  [197] = {x=-25.429863, y=27.236716, z=96.648372, rx=-178.000688, ry=-0.000306, rz=-0.000289, shoulder=lefty, elbow=epositive, wrist=wpositive, fatherId=frmaster[2]}
  [198] = {x=-24.431312, y=27.249472, z=96.640619, rx=-177.999992, ry=-0.000305, rz=0.000037, shoulder=lefty, elbow=epositive, wrist=wpositive, fatherId=frmaster[2]}
  [199] = {x=-23.439357, y=27.256646, z=96.642496, rx=-178.000278, ry=-0.00008, rz=0.00033, shoulder=lefty, elbow=epositive, wrist=wpositive, fatherId=frmaster[2]}
  [200] = {x=-22.438851, y=27.268013, z=96.64425, rx=-178.000546, ry=0.000117, rz=-0.000381, shoulder=lefty, elbow=epositive, wrist=wpositive, fatherId=frmaster[2]}
  [201] = {x=-21.43819, y=27.28289, z=96.645991, rx=-177.999822, ry=0.000137, rz=-0.000095, shoulder=lefty, elbow=epositive, wrist=wpositive, fatherId=frmaster[2]}
  [202] = {x=-20.443726, y=27.289844, z=96.648903, rx=-178.001063, ry=0.000565, rz=0.000171, shoulder=lefty, elbow=epositive, wrist=wpositive, fatherId=frmaster[2]}
  [203] = {x=-19.450271, y=27.300156, z=96.643398, rx=-178.000499, ry=-0.00027, rz=0.00003, shoulder=lefty, elbow=epositive, wrist=wpositive, fatherId=frmaster[2]}
  [204] = {x=-18.446659, y=27.31259, z=96.642606, rx=-177.999749, ry=-0.000237, rz=-0.000711, shoulder=lefty, elbow=epositive, wrist=wpositive, fatherId=frmaster[2]}
  [205] = {x=-17.450599, y=27.324153, z=96.641778, rx=-177.999982, ry=0.000019, rz=-0.000456, shoulder=lefty, elbow=epositive, wrist=wpositive, fatherId=frmaster[2]}
  [206] = {x=-16.452954, y=27.332175, z=96.642123, rx=-178.000204, ry=0.000286, rz=-0.000221, shoulder=lefty, elbow=epositive, wrist=wpositive, fatherId=frmaster[2]}
  [207] = {x=-15.456767, y=27.345858, z=96.637596, rx=-177.999612, ry=-0.000534, rz=-0.00039, shoulder=lefty, elbow=epositive, wrist=wpositive, fatherId=frmaster[2]}
  [208] = {x=-14.4578, y=27.356168, z=96.642655, rx=-177.999817, ry=-0.000253, rz=-0.000178, shoulder=lefty, elbow=epositive, wrist=wpositive, fatherId=frmaster[2]}
  [209] = {x=-13.46591, y=27.363257, z=96.644106, rx=-178.00002, ry=0.000066, rz=0.000029, shoulder=lefty, elbow=epositive, wrist=wpositive, fatherId=frmaster[2]}
  [210] = {x=-12.465449, y=27.37475, z=96.645422, rx=-178.000206, ry=0.000355, rz=0.000232, shoulder=lefty, elbow=epositive, wrist=wpositive, fatherId=frmaster[2]}
  [211] = {x=-11.465766, y=27.388433, z=96.638237, rx=-177.999587, ry=-0.000451, rz=-0.000966, shoulder=lefty, elbow=epositive, wrist=wpositive, fatherId=frmaster[2]}
  [212] = {x=-10.471416, y=27.396685, z=96.64071, rx=-177.999763, ry=-0.000114, rz=0.000213, shoulder=lefty, elbow=epositive, wrist=wpositive, fatherId=frmaster[2]}
  [213] = {x=-9.476659, y=27.407266, z=96.643115, rx=-177.99993, ry=0.000228, rz=0.000387, shoulder=lefty, elbow=epositive, wrist=wpositive, fatherId=frmaster[2]}
  [214] = {x=-8.473698, y=27.418659, z=96.641745, rx=-178.000267, ry=-0.000352, rz=-0.000853, shoulder=lefty, elbow=epositive, wrist=wpositive, fatherId=frmaster[2]}
  [215] = {x=-7.476841, y=27.428148, z=96.645231, rx=-178.000415, ry=0.000004, rz=-0.000703, shoulder=lefty, elbow=epositive, wrist=wpositive, fatherId=frmaster[2]}
  [216] = {x=-6.479573, y=27.439988, z=96.648645, rx=-178.000553, ry=0.000365, rz=-0.000557, shoulder=lefty, elbow=epositive, wrist=wpositive, fatherId=frmaster[2]}
  [217] = {x=-5.482244, y=27.450503, z=96.648342, rx=-178.000876, ry=-0.000161, rz=-0.000826, shoulder=lefty, elbow=epositive, wrist=wpositive, fatherId=frmaster[2]}
  [218] = {x=-4.49109, y=27.459137, z=96.644439, rx=-178.000029, ry=0.000027, rz=0.000311, shoulder=lefty, elbow=epositive, wrist=wpositive, fatherId=frmaster[2]}
  [219] = {x=-3.491358, y=27.47236, z=96.640386, rx=-177.999165, ry=0.000182, rz=0.000444, shoulder=lefty, elbow=epositive, wrist=wpositive, fatherId=frmaster[2]}
  [220] = {x=-2.491458, y=27.484219, z=96.641061, rx=-177.999465, ry=-0.000328, rz=-0.000853, shoulder=lefty, elbow=epositive, wrist=wpositive, fatherId=frmaster[2]}
  [221] = {x=-1.497362, y=27.492926, z=96.646554, rx=-178.000541, ry=0.000317, rz=0.000238, shoulder=lefty, elbow=epositive, wrist=wpositive, fatherId=frmaster[2]}
  [222] = {x=-0.495266, y=27.503824, z=96.648283, rx=-178.000826, ry=-0.000176, rz=-0.001082, shoulder=lefty, elbow=epositive, wrist=wpositive, fatherId=frmaster[2]}
  [223] = {x=0.500089, y=27.515119, z=96.641527, rx=-177.999935, ry=0.000028, rz=0.000016, shoulder=lefty, elbow=epositive, wrist=wpositive, fatherId=frmaster[2]}
  [224] = {x=1.495371, y=27.526248, z=96.639538, rx=-177.99924, ry=-0.000651, rz=-0.000313, shoulder=lefty, elbow=epositive, wrist=wpositive, fatherId=frmaster[2]}
  [225] = {x=2.49304, y=27.536538, z=96.642297, rx=-177.999304, ry=-0.000205, rz=-0.000256, shoulder=lefty, elbow=epositive, wrist=wpositive, fatherId=frmaster[2]}
  [226] = {x=3.491932, y=27.545823, z=96.641306, rx=-177.999358, ry=0.000245, rz=-0.000205, shoulder=lefty, elbow=epositive, wrist=wpositive, fatherId=frmaster[2]}
  [227] = {x=4.490166, y=27.557254, z=96.640215, rx=-177.999614, ry=-0.00019, rz=-0.000562, shoulder=lefty, elbow=epositive, wrist=wpositive, fatherId=frmaster[2]}
  [228] = {x=5.482361, y=27.566672, z=96.643983, rx=-177.999657, ry=0.000308, rz=0.000462, shoulder=lefty, elbow=epositive, wrist=wpositive, fatherId=frmaster[2]}
  [229] = {x=6.482875, y=27.57725, z=96.643913, rx=-177.999897, ry=-0.000112, rz=0.00008, shoulder=lefty, elbow=epositive, wrist=wpositive, fatherId=frmaster[2]}
  [230] = {x=7.476743, y=27.588075, z=96.643826, rx=-177.999922, ry=0.000394, rz=0.000095, shoulder=lefty, elbow=epositive, wrist=wpositive, fatherId=frmaster[2]}
  [231] = {x=8.478648, y=27.6013, z=96.639929, rx=-177.999177, ry=-0.000259, rz=-0.000296, shoulder=lefty, elbow=epositive, wrist=wpositive, fatherId=frmaster[2]}
  [232] = {x=9.473739, y=27.611047, z=96.640839, rx=-177.999403, ry=-0.000629, rz=-0.000709, shoulder=lefty, elbow=epositive, wrist=wpositive, fatherId=frmaster[2]}
  [233] = {x=10.471276, y=27.620049, z=96.646501, rx=-178.000369, ry=0.000144, rz=0.000258, shoulder=lefty, elbow=epositive, wrist=wpositive, fatherId=frmaster[2]}
  [234] = {x=11.467775, y=27.632457, z=96.64357, rx=-177.999611, ry=-0.000461, rz=-0.000163, shoulder=lefty, elbow=epositive, wrist=wpositive, fatherId=frmaster[2]}
  [235] = {x=12.467578, y=27.640793, z=96.641696, rx=-177.999588, ry=0.000076, rz=-0.000206, shoulder=lefty, elbow=epositive, wrist=wpositive, fatherId=frmaster[2]}
  [236] = {x=13.465879, y=27.654652, z=96.643403, rx=-177.999783, ry=-0.000272, rz=-0.000653, shoulder=lefty, elbow=epositive, wrist=wpositive, fatherId=frmaster[2]}
  [237] = {x=14.459037, y=27.663095, z=96.646276, rx=-177.999749, ry=0.000314, rz=0.000276, shoulder=lefty, elbow=epositive, wrist=wpositive, fatherId=frmaster[2]}
  [238] = {x=15.460577, y=27.672929, z=96.645267, rx=-177.999927, ry=-0.00002, rz=-0.000198, shoulder=lefty, elbow=epositive, wrist=wpositive, fatherId=frmaster[2]}
  [239] = {x=16.454396, y=27.682636, z=96.644215, rx=-178.000108, ry=-0.000315, rz=0.000324, shoulder=lefty, elbow=epositive, wrist=wpositive, fatherId=frmaster[2]}
  [240] = {x=17.450704, y=27.691678, z=96.647917, rx=-178.001011, ry=0.000544, rz=0.000221, shoulder=lefty, elbow=epositive, wrist=wpositive, fatherId=frmaster[2]}
  [241] = {x=18.445962, y=27.704133, z=96.642978, rx=-178.00021, ry=-0.000001, rz=0.000733, shoulder=lefty, elbow=epositive, wrist=wpositive, fatherId=frmaster[2]}
  [242] = {x=19.44329, y=27.713454, z=96.647675, rx=-178.000365, ry=-0.000271, rz=0.000207, shoulder=lefty, elbow=epositive, wrist=wpositive, fatherId=frmaster[2]}
  [243] = {x=20.442373, y=27.724431, z=96.643656, rx=-178.000275, ry=0.000342, rz=0.000087, shoulder=lefty, elbow=epositive, wrist=wpositive, fatherId=frmaster[2]}
  [244] = {x=21.441478, y=27.7354, z=96.644408, rx=-178.000414, ry=0.000079, rz=-0.000449, shoulder=lefty, elbow=epositive, wrist=wpositive, fatherId=frmaster[2]}
  [245] = {x=22.441019, y=27.74886, z=96.645044, rx=-178.000548, ry=-0.000181, rz=0.000011, shoulder=lefty, elbow=epositive, wrist=wpositive, fatherId=frmaster[2]}
  [246] = {x=23.435503, y=27.756909, z=96.646817, rx=-178.000434, ry=0.00049, rz=-0.000161, shoulder=lefty, elbow=epositive, wrist=wpositive, fatherId=frmaster[2]}
  [247] = {x=24.437414, y=27.769943, z=96.639796, rx=-177.999589, ry=-0.000032, rz=-0.000711, shoulder=lefty, elbow=epositive, wrist=wpositive, fatherId=frmaster[2]}
  [248] = {x=25.432704, y=27.779323, z=96.646183, rx=-178.000668, ry=0.000036, rz=-0.000302, shoulder=lefty, elbow=epositive, wrist=wpositive, fatherId=frmaster[2]}
  [249] = {x=26.429026, y=27.789092, z=96.648755, rx=-178.000776, ry=-0.000162, rz=0.000103, shoulder=lefty, elbow=epositive, wrist=wpositive, fatherId=frmaster[2]}
  [250] = {x=27.426778, y=27.801741, z=96.642603, rx=-177.999665, ry=0.000247, rz=-0.000091, shoulder=lefty, elbow=epositive, wrist=wpositive, fatherId=frmaster[2]}
  [251] = {x=28.424908, y=27.813257, z=96.641179, rx=-177.999759, ry=0.000054, rz=-0.000696, shoulder=lefty, elbow=epositive, wrist=wpositive, fatherId=frmaster[2]}
  [252] = {x=29.416007, y=27.822315, z=96.644609, rx=-177.999852, ry=-0.000095, rz=0.000675, shoulder=lefty, elbow=epositive, wrist=wpositive, fatherId=frmaster[2]}
  [253] = {x=30.416648, y=27.833458, z=96.644092, rx=-177.99993, ry=-0.000274, rz=0.000042, shoulder=lefty, elbow=epositive, wrist=wpositive, fatherId=frmaster[2]}
  [254] = {x=31.410613, y=27.840971, z=96.648389, rx=-178.000966, ry=-0.000127, rz=0.000385, shoulder=lefty, elbow=epositive, wrist=wpositive, fatherId=frmaster[2]}
  [255] = {x=32.413819, y=27.855441, z=96.6439, rx=-177.999808, ry=0.000303, rz=0.000128, shoulder=lefty, elbow=epositive, wrist=wpositive, fatherId=frmaster[2]}
  [256] = {x=33.40927, y=27.865955, z=96.64421, rx=-177.999869, ry=0.000174, rz=0.000461, shoulder=lefty, elbow=epositive, wrist=wpositive, fatherId=frmaster[2]}
  [257] = {x=34.406123, y=27.875773, z=96.640614, rx=-177.999923, ry=0.000048, rz=-0.000211, shoulder=lefty, elbow=epositive, wrist=wpositive, fatherId=frmaster[2]}
  [258] = {x=35.404123, y=27.886022, z=96.641803, rx=-177.999968, ry=-0.000067, rz=0.000093, shoulder=lefty, elbow=epositive, wrist=wpositive, fatherId=frmaster[2]}
  [259] = {x=36.403626, y=27.895551, z=96.647741, rx=-178.00096, ry=0.000119, rz=-0.000625, shoulder=lefty, elbow=epositive, wrist=wpositive, fatherId=frmaster[2]}
  [260] = {x=37.394959, y=27.905922, z=96.644981, rx=-178.000043, ry=-0.000248, rz=0.000669, shoulder=lefty, elbow=epositive, wrist=wpositive, fatherId=frmaster[2]}
  [261] = {x=38.395954, y=27.918548, z=96.646901, rx=-178.000064, ry=-0.000347, rz=-0.00006, shoulder=lefty, elbow=epositive, wrist=wpositive, fatherId=frmaster[2]}
  [262] = {x=39.390215, y=27.927562, z=96.644957, rx=-178.000087, ry=-0.000409, rz=0.000205, shoulder=lefty, elbow=epositive, wrist=wpositive, fatherId=frmaster[2]}
  [263] = {x=40.387074, y=27.936225, z=96.64777, rx=-178.000778, ry=0.000721, rz=0.000825, shoulder=lefty, elbow=epositive, wrist=wpositive, fatherId=frmaster[2]}
  [264] = {x=41.390983, y=27.9514, z=96.641707, rx=-177.999821, ry=0.000332, rz=0.00008, shoulder=lefty, elbow=epositive, wrist=wpositive, fatherId=frmaster[2]}
  [265] = {x=42.388987, y=27.960812, z=96.645394, rx=-177.999816, ry=0.000292, rz=-0.000708, shoulder=lefty, elbow=epositive, wrist=wpositive, fatherId=frmaster[2]}
  [266] = {x=43.379636, y=27.968603, z=96.648958, rx=-178.000764, ry=0.000594, rz=0.000497, shoulder=lefty, elbow=epositive, wrist=wpositive, fatherId=frmaster[2]}
  [267] = {x=44.379508, y=27.98005, z=96.64854, rx=-178.000744, ry=0.000562, rz=-0.000302, shoulder=lefty, elbow=epositive, wrist=wpositive, fatherId=frmaster[2]}
  [268] = {x=45.380448, y=27.992117, z=96.644193, rx=-177.999765, ry=0.000225, rz=-0.000107, shoulder=lefty, elbow=epositive, wrist=wpositive, fatherId=frmaster[2]}
  [269] = {x=46.374032, y=28.002542, z=96.63971, rx=-177.999739, ry=0.000231, rz=0.000082, shoulder=lefty, elbow=epositive, wrist=wpositive, fatherId=frmaster[2]}
  [270] = {x=47.369898, y=28.010305, z=96.644922, rx=-178.000651, ry=0.000565, rz=0.000229, shoulder=lefty, elbow=epositive, wrist=wpositive, fatherId=frmaster[2]}
  [271] = {x=48.365713, y=28.021921, z=96.641283, rx=-177.999657, ry=0.000272, rz=0.000388, shoulder=lefty, elbow=epositive, wrist=wpositive, fatherId=frmaster[2]}
  [272] = {x=49.363071, y=28.03297, z=96.642392, rx=-177.999604, ry=0.0003, rz=0.000523, shoulder=lefty, elbow=epositive, wrist=wpositive, fatherId=frmaster[2]}
  [273] = {x=50.361979, y=28.043473, z=96.648253, rx=-178.00049, ry=0.000655, rz=0.000633, shoulder=lefty, elbow=epositive, wrist=wpositive, fatherId=frmaster[2]}
  [274] = {x=51.360884, y=28.054305, z=96.650146, rx=-178.000715, ry=-0.000184, rz=-0.000633, shoulder=lefty, elbow=epositive, wrist=wpositive, fatherId=frmaster[2]}
  [275] = {x=52.35303, y=28.065007, z=96.643192, rx=-177.999702, ry=-0.000433, rz=0.000485, shoulder=lefty, elbow=epositive, wrist=wpositive, fatherId=frmaster[2]}
  [276] = {x=53.356032, y=28.075245, z=96.645837, rx=-178.000563, ry=-0.000058, rz=-0.00044, shoulder=lefty, elbow=epositive, wrist=wpositive, fatherId=frmaster[2]}
  [277] = {x=54.350898, y=28.086084, z=96.648419, rx=-178.000477, ry=0.000033, rz=-0.000372, shoulder=lefty, elbow=epositive, wrist=wpositive, fatherId=frmaster[2]}
  [278] = {x=55.34723, y=28.096492, z=96.646978, rx=-178.000384, ry=0.000126, rz=0.00069, shoulder=lefty, elbow=epositive, wrist=wpositive, fatherId=frmaster[2]}
  [279] = {x=56.344633, y=28.107643, z=96.641542, rx=-177.999339, ry=-0.000106, rz=0.000746, shoulder=lefty, elbow=epositive, wrist=wpositive, fatherId=frmaster[2]}
  [280] = {x=57.344096, y=28.117134, z=96.649602, rx=-178.001114, ry=0.000662, rz=-0.000242, shoulder=lefty, elbow=epositive, wrist=wpositive, fatherId=frmaster[2]}
  [281] = {x=58.342965, y=28.131764, z=96.639977, rx=-177.999111, ry=0.000102, rz=-0.000198, shoulder=lefty, elbow=epositive, wrist=wpositive, fatherId=frmaster[2]}
  [282] = {x=59.335845, y=28.137903, z=96.648846, rx=-178.001185, ry=0.000045, rz=0.000419, shoulder=lefty, elbow=epositive, wrist=wpositive, fatherId=frmaster[2]}
  [283] = {x=60.337345, y=28.152913, z=96.639946, rx=-177.999168, ry=-0.000511, rz=-0.000567, shoulder=lefty, elbow=epositive, wrist=wpositive, fatherId=frmaster[2]}
  [284] = {x=61.332762, y=28.162955, z=96.644632, rx=-177.999974, ry=-0.000014, rz=0.0004, shoulder=lefty, elbow=epositive, wrist=wpositive, fatherId=frmaster[2]}
  [285] = {x=62.33034, y=28.170761, z=96.641412, rx=-177.99983, ry=0.00015, rz=0.000362, shoulder=lefty, elbow=epositive, wrist=wpositive, fatherId=frmaster[2]}
  [286] = {x=63.328401, y=28.181264, z=96.646825, rx=-178.000617, ry=0.000663, rz=0.000298, shoulder=lefty, elbow=epositive, wrist=wpositive, fatherId=frmaster[2]}
  [287] = {x=64.326455, y=28.192238, z=96.648189, rx=-178.000773, ry=-0.000038, rz=-0.000131, shoulder=lefty, elbow=epositive, wrist=wpositive, fatherId=frmaster[2]}
  [288] = {x=65.317712, y=28.202973, z=96.640597, rx=-177.999677, ry=-0.000175, rz=0.000812, shoulder=lefty, elbow=epositive, wrist=wpositive, fatherId=frmaster[2]}
  [289] = {x=66.319474, y=28.21489, z=96.642673, rx=-177.999499, ry=0.000011, rz=-0.00029, shoulder=lefty, elbow=epositive, wrist=wpositive, fatherId=frmaster[2]}
  [290] = {x=67.314662, y=28.223041, z=96.649572, rx=-178.000257, ry=0.000587, rz=0.00058, shoulder=lefty, elbow=epositive, wrist=wpositive, fatherId=frmaster[2]}
  [291] = {x=66.315693, y=28.224826, z=96.640494, rx=-177.999504, ry=-0.000003, rz=0.00075, shoulder=lefty, elbow=epositive, wrist=wpositive, fatherId=frmaster[2]}
  [292] = {x=65.319102, y=28.224406, z=96.641152, rx=-177.999677, ry=-0.00023, rz=-0.000128, shoulder=lefty, elbow=epositive, wrist=wpositive, fatherId=frmaster[2]}
  [293] = {x=64.324104, y=28.22369, z=96.646545, rx=-178.000779, ry=-0.000107, rz=-0.000031, shoulder=lefty, elbow=epositive, wrist=wpositive, fatherId=frmaster[2]}
  [294] = {x=63.330069, y=28.227356, z=96.642947, rx=-177.999679, ry=0.000206, rz=-0.000563, shoulder=lefty, elbow=epositive, wrist=wpositive, fatherId=frmaster[2]}
  [295] = {x=62.329597, y=28.223791, z=96.649083, rx=-178.000774, ry=0.000371, rz=0.000502, shoulder=lefty, elbow=epositive, wrist=wpositive, fatherId=frmaster[2]}
  [296] = {x=61.329025, y=28.224226, z=96.646232, rx=-177.999982, ry=-0.000146, rz=0.000579, shoulder=lefty, elbow=epositive, wrist=wpositive, fatherId=frmaster[2]}
  [297] = {x=60.338108, y=28.227749, z=96.639243, rx=-177.999172, ry=-0.00069, rz=-0.00035, shoulder=lefty, elbow=epositive, wrist=wpositive, fatherId=frmaster[2]}
  [298] = {x=59.3418, y=28.227852, z=96.645882, rx=-177.999933, ry=0.000363, rz=0.000039, shoulder=lefty, elbow=epositive, wrist=wpositive, fatherId=frmaster[2]}
  [299] = {x=58.337267, y=28.22513, z=96.639746, rx=-177.999123, ry=-0.000099, rz=0.000078, shoulder=lefty, elbow=epositive, wrist=wpositive, fatherId=frmaster[2]}
  [300] = {x=57.342568, y=28.225297, z=96.647079, rx=-178.000179, ry=0.000084, rz=0.000072, shoulder=lefty, elbow=epositive, wrist=wpositive, fatherId=frmaster[2]}
  [301] = {x=56.349269, y=28.225156, z=96.641568, rx=-178.000286, ry=-0.000069, rz=0.00008, shoulder=lefty, elbow=epositive, wrist=wpositive, fatherId=frmaster[2]}
  [302] = {x=55.347937, y=28.225548, z=96.644761, rx=-178.000392, ry=-0.000178, rz=0.000061, shoulder=lefty, elbow=epositive, wrist=wpositive, fatherId=frmaster[2]}
  [303] = {x=54.348862, y=28.223565, z=96.648874, rx=-178.000488, ry=-0.000279, rz=0.000017, shoulder=lefty, elbow=epositive, wrist=wpositive, fatherId=frmaster[2]}
  [304] = {x=53.351594, y=28.223574, z=96.644005, rx=-178.000278, ry=0.000496, rz=0.000355, shoulder=lefty, elbow=epositive, wrist=wpositive, fatherId=frmaster[2]}
  [305] = {x=52.354048, y=28.225066, z=96.643944, rx=-177.999413, ry=0.000081, rz=0.0003, shoulder=lefty, elbow=epositive, wrist=wpositive, fatherId=frmaster[2]}
  [306] = {x=51.358385, y=28.224976, z=96.639825, rx=-177.999488, ry=-0.00001, rz=0.000239, shoulder=lefty, elbow=epositive, wrist=wpositive, fatherId=frmaster[2]}
  [307] = {x=50.36391, y=28.22554, z=96.640487, rx=-177.999552, ry=-0.000092, rz=0.000153, shoulder=lefty, elbow=epositive, wrist=wpositive, fatherId=frmaster[2]}
  [308] = {x=49.362859, y=28.222403, z=96.645949, rx=-178.000563, ry=0.000186, rz=0.000041, shoulder=lefty, elbow=epositive, wrist=wpositive, fatherId=frmaster[2]}
  [309] = {x=48.369924, y=28.22634, z=96.642469, rx=-177.999663, ry=-0.000206, rz=-0.000056, shoulder=lefty, elbow=epositive, wrist=wpositive, fatherId=frmaster[2]}
  [310] = {x=47.370415, y=28.226583, z=96.643793, rx=-177.999711, ry=-0.000238, rz=-0.000179, shoulder=lefty, elbow=epositive, wrist=wpositive, fatherId=frmaster[2]}
  [311] = {x=46.373506, y=28.22312, z=96.646033, rx=-178.0007, ry=0.000049, rz=-0.000327, shoulder=lefty, elbow=epositive, wrist=wpositive, fatherId=frmaster[2]}
  [312] = {x=45.376662, y=28.223474, z=96.648142, rx=-178.000731, ry=0.000027, rz=-0.000481, shoulder=lefty, elbow=epositive, wrist=wpositive, fatherId=frmaster[2]}
  [313] = {x=44.380179, y=28.226543, z=96.641372, rx=-177.999805, ry=-0.000306, rz=-0.000621, shoulder=lefty, elbow=epositive, wrist=wpositive, fatherId=frmaster[2]}
  [314] = {x=43.377846, y=28.223871, z=96.644349, rx=-177.999827, ry=-0.00028, rz=0.000195, shoulder=lefty, elbow=epositive, wrist=wpositive, fatherId=frmaster[2]}
  [315] = {x=42.384028, y=28.226973, z=96.638395, rx=-177.998882, ry=-0.000594, rz=0.000025, shoulder=lefty, elbow=epositive, wrist=wpositive, fatherId=frmaster[2]}
  [316] = {x=41.384715, y=28.223153, z=96.642144, rx=-177.99984, ry=-0.000252, rz=-0.000189, shoulder=lefty, elbow=epositive, wrist=wpositive, fatherId=frmaster[2]}
  [317] = {x=40.394003, y=28.224982, z=96.645661, rx=-178.000784, ry=0.000055, rz=-0.000407, shoulder=lefty, elbow=epositive, wrist=wpositive, fatherId=frmaster[2]}
  [318] = {x=39.396232, y=28.224365, z=96.645335, rx=-178.000775, ry=0.000099, rz=-0.000632, shoulder=lefty, elbow=epositive, wrist=wpositive, fatherId=frmaster[2]}
  [319] = {x=38.39856, y=28.227533, z=96.644894, rx=-177.999803, ry=-0.000151, rz=-0.000862, shoulder=lefty, elbow=epositive, wrist=wpositive, fatherId=frmaster[2]}
  [320] = {x=37.395633, y=28.222683, z=96.64543, rx=-178.000741, ry=0.000235, rz=-0.000116, shoulder=lefty, elbow=epositive, wrist=wpositive, fatherId=frmaster[2]}
  [321] = {x=36.4006, y=28.225741, z=96.645829, rx=-177.999752, ry=0.000002, rz=-0.000375, shoulder=lefty, elbow=epositive, wrist=wpositive, fatherId=frmaster[2]}
  [322] = {x=35.407371, y=28.226988, z=96.642262, rx=-177.999711, ry=0.000067, rz=-0.000639, shoulder=lefty, elbow=epositive, wrist=wpositive, fatherId=frmaster[2]}
  [323] = {x=34.407167, y=28.225766, z=96.64354, rx=-177.99967, ry=0.000175, rz=0.000073, shoulder=lefty, elbow=epositive, wrist=wpositive, fatherId=frmaster[2]}
  [324] = {x=33.408488, y=28.223834, z=96.649546, rx=-178.000577, ry=0.00058, rz=0.000761, shoulder=lefty, elbow=epositive, wrist=wpositive, fatherId=frmaster[2]}
  [325] = {x=32.409104, y=28.224226, z=96.646752, rx=-178.000784, ry=-0.000191, rz=0.000076, shoulder=lefty, elbow=epositive, wrist=wpositive, fatherId=frmaster[2]}
  [326] = {x=31.411883, y=28.225438, z=96.640112, rx=-177.999761, ry=-0.000358, rz=-0.000228, shoulder=lefty, elbow=epositive, wrist=wpositive, fatherId=frmaster[2]}
  [327] = {x=30.416178, y=28.225894, z=96.638211, rx=-177.999687, ry=-0.00023, rz=0.000444, shoulder=lefty, elbow=epositive, wrist=wpositive, fatherId=frmaster[2]}
  [328] = {x=29.42164, y=28.226746, z=96.641083, rx=-177.999604, ry=-0.000092, rz=0.000093, shoulder=lefty, elbow=epositive, wrist=wpositive, fatherId=frmaster[2]}
  [329] = {x=28.420364, y=28.224059, z=96.640136, rx=-177.999523, ry=0.000084, rz=0.000737, shoulder=lefty, elbow=epositive, wrist=wpositive, fatherId=frmaster[2]}
  [330] = {x=27.427709, y=28.226726, z=96.638986, rx=-177.999426, ry=0.000229, rz=0.000376, shoulder=lefty, elbow=epositive, wrist=wpositive, fatherId=frmaster[2]}
  [331] = {x=26.426984, y=28.226665, z=96.642663, rx=-177.99958, ry=-0.000466, rz=-0.000398, shoulder=lefty, elbow=epositive, wrist=wpositive, fatherId=frmaster[2]}
  [332] = {x=25.428743, y=28.226172, z=96.642478, rx=-177.999474, ry=-0.000274, rz=0.000212, shoulder=lefty, elbow=epositive, wrist=wpositive, fatherId=frmaster[2]}
  [333] = {x=24.431987, y=28.224856, z=96.647023, rx=-178.000322, ry=0.0002, rz=-0.000199, shoulder=lefty, elbow=epositive, wrist=wpositive, fatherId=frmaster[2]}
  [334] = {x=23.436288, y=28.223936, z=96.647748, rx=-178.0002, ry=0.000405, rz=0.000384, shoulder=lefty, elbow=epositive, wrist=wpositive, fatherId=frmaster[2]}
  [335] = {x=22.439977, y=28.225228, z=96.648333, rx=-178.000316, ry=-0.000273, rz=-0.000431, shoulder=lefty, elbow=epositive, wrist=wpositive, fatherId=frmaster[2]}
  [336] = {x=21.43798, y=28.223331, z=96.645149, rx=-178.000188, ry=-0.000027, rz=0.000141, shoulder=lefty, elbow=epositive, wrist=wpositive, fatherId=frmaster[2]}
  [337] = {x=20.445275, y=28.224428, z=96.646671, rx=-178.000043, ry=0.000196, rz=-0.000307, shoulder=lefty, elbow=epositive, wrist=wpositive, fatherId=frmaster[2]}
  [338] = {x=19.443722, y=28.22513, z=96.63956, rx=-177.999174, ry=-0.000699, rz=-0.00014, shoulder=lefty, elbow=epositive, wrist=wpositive, fatherId=frmaster[2]}
  [339] = {x=18.452949, y=28.22782, z=96.645686, rx=-177.999977, ry=-0.000201, rz=-0.000616, shoulder=lefty, elbow=epositive, wrist=wpositive, fatherId=frmaster[2]}
  [340] = {x=17.454983, y=28.228271, z=96.639534, rx=-177.998851, ry=-0.000191, rz=-0.00008, shoulder=lefty, elbow=epositive, wrist=wpositive, fatherId=frmaster[2]}
  [341] = {x=16.45855, y=28.227744, z=96.646665, rx=-177.999648, ry=0.000351, rz=-0.000583, shoulder=lefty, elbow=epositive, wrist=wpositive, fatherId=frmaster[2]}
  [342] = {x=15.454136, y=28.22355, z=96.641488, rx=-177.999714, ry=-0.00022, rz=0.000527, shoulder=lefty, elbow=epositive, wrist=wpositive, fatherId=frmaster[2]}
  [343] = {x=14.459207, y=28.225825, z=96.644722, rx=-177.99953, ry=0.000072, rz=0.000015, shoulder=lefty, elbow=epositive, wrist=wpositive, fatherId=frmaster[2]}
  [344] = {x=13.464838, y=28.225749, z=96.644096, rx=-178.000535, ry=-0.00027, rz=-0.000902, shoulder=lefty, elbow=epositive, wrist=wpositive, fatherId=frmaster[2]}
  [345] = {x=12.464123, y=28.224881, z=96.63983, rx=-177.999376, ry=-0.000185, rz=0.000575, shoulder=lefty, elbow=epositive, wrist=wpositive, fatherId=frmaster[2]}
  [346] = {x=11.473359, y=28.224322, z=96.648709, rx=-178.001104, ry=0.000624, rz=0.000015, shoulder=lefty, elbow=epositive, wrist=wpositive, fatherId=frmaster[2]}
  [347] = {x=10.47335, y=28.224739, z=96.640534, rx=-178.000154, ry=-0.00017, rz=0.000082, shoulder=lefty, elbow=epositive, wrist=wpositive, fatherId=frmaster[2]}
  [348] = {x=9.47562, y=28.225569, z=96.645657, rx=-177.999939, ry=0.000188, rz=-0.000488, shoulder=lefty, elbow=epositive, wrist=wpositive, fatherId=frmaster[2]}
  [349] = {x=8.478405, y=28.224016, z=96.646942, rx=-178.000907, ry=-0.000099, rz=-0.000465, shoulder=lefty, elbow=epositive, wrist=wpositive, fatherId=frmaster[2]}
  [350] = {x=7.482363, y=28.226424, z=96.639671, rx=-177.999708, ry=0.00002, rz=-0.000027, shoulder=lefty, elbow=epositive, wrist=wpositive, fatherId=frmaster[2]}
  [351] = {x=6.478268, y=28.226242, z=96.645728, rx=-177.999694, ry=-0.000459, rz=-0.000031, shoulder=lefty, elbow=epositive, wrist=wpositive, fatherId=frmaster[2]}
  [352] = {x=5.484899, y=28.226678, z=96.639421, rx=-177.999449, ry=-0.000085, rz=0.000381, shoulder=lefty, elbow=epositive, wrist=wpositive, fatherId=frmaster[2]}
  [353] = {x=4.483458, y=28.22453, z=96.646432, rx=-178.000387, ry=-0.000317, rz=0.00035, shoulder=lefty, elbow=epositive, wrist=wpositive, fatherId=frmaster[2]}
  [354] = {x=3.492522, y=28.224047, z=96.649621, rx=-178.001098, ry=0.000307, rz=-0.00028, shoulder=lefty, elbow=epositive, wrist=wpositive, fatherId=frmaster[2]}
  [355] = {x=2.492441, y=28.224601, z=96.644333, rx=-178.000075, ry=-0.000387, rz=-0.000304, shoulder=lefty, elbow=epositive, wrist=wpositive, fatherId=frmaster[2]}
  [356] = {x=1.494795, y=28.224353, z=96.643784, rx=-177.999807, ry=0.000048, rz=0.000057, shoulder=lefty, elbow=epositive, wrist=wpositive, fatherId=frmaster[2]}
  [357] = {x=0.496527, y=28.226268, z=96.643131, rx=-177.999738, ry=-0.000402, rz=0.000007, shoulder=lefty, elbow=epositive, wrist=wpositive, fatherId=frmaster[2]}
  [358] = {x=-0.498539, y=28.223928, z=96.643567, rx=-178.000429, ry=0.000272, rz=0.000344, shoulder=lefty, elbow=epositive, wrist=wpositive, fatherId=frmaster[2]}
  [359] = {x=-1.49451, y=28.224924, z=96.643944, rx=-178.000341, ry=-0.000165, rz=-0.000733, shoulder=lefty, elbow=epositive, wrist=wpositive, fatherId=frmaster[2]}
  [360] = {x=-2.496228, y=28.222784, z=96.649121, rx=-178.001026, ry=0.000552, rz=0.000579, shoulder=lefty, elbow=epositive, wrist=wpositive, fatherId=frmaster[2]}
  [361] = {x=-3.490776, y=28.226328, z=96.64572, rx=-177.999944, ry=-0.000095, rz=-0.000507, shoulder=lefty, elbow=epositive, wrist=wpositive, fatherId=frmaster[2]}
  [362] = {x=-4.491413, y=28.223063, z=96.643481, rx=-177.999836, ry=-0.000478, rz=0.000386, shoulder=lefty, elbow=epositive, wrist=wpositive, fatherId=frmaster[2]}
  [363] = {x=-5.482276, y=28.224579, z=96.649538, rx=-178.00049, ry=0.000219, rz=-0.00033, shoulder=lefty, elbow=epositive, wrist=wpositive, fatherId=frmaster[2]}
  [364] = {x=-6.482094, y=28.226153, z=96.638695, rx=-177.999388, ry=-0.000376, rz=-0.00043, shoulder=lefty, elbow=epositive, wrist=wpositive, fatherId=frmaster[2]}
  [365] = {x=-7.478889, y=28.224423, z=96.645871, rx=-178.000037, ry=0.000366, rz=-0.00017, shoulder=lefty, elbow=epositive, wrist=wpositive, fatherId=frmaster[2]}
  [366] = {x=-8.476412, y=28.224902, z=96.644525, rx=-177.999892, ry=0.000005, rz=-0.000311, shoulder=lefty, elbow=epositive, wrist=wpositive, fatherId=frmaster[2]}
  [367] = {x=-9.472672, y=28.224216, z=96.647902, rx=-178.000715, ry=-0.000141, rz=-0.000473, shoulder=lefty, elbow=epositive, wrist=wpositive, fatherId=frmaster[2]}
  [368] = {x=-10.467732, y=28.227381, z=96.642829, rx=-177.999388, ry=0.000192, rz=-0.000209, shoulder=lefty, elbow=epositive, wrist=wpositive, fatherId=frmaster[2]}
  [369] = {x=-11.469983, y=28.223475, z=96.647344, rx=-178.000202, ry=0.000092, rz=0.000605, shoulder=lefty, elbow=epositive, wrist=wpositive, fatherId=frmaster[2]}
  [370] = {x=-12.46373, y=28.22411, z=96.643303, rx=-178.00002, ry=-0.000248, rz=-0.00057, shoulder=lefty, elbow=epositive, wrist=wpositive, fatherId=frmaster[2]}
  [371] = {x=-13.464097, y=28.225225, z=96.639265, rx=-177.999658, ry=0.000343, rz=0.000666, shoulder=lefty, elbow=epositive, wrist=wpositive, fatherId=frmaster[2]}
  [372] = {x=-14.46379, y=28.222571, z=96.644783, rx=-178.000445, ry=0.000255, rz=0.000452, shoulder=lefty, elbow=epositive, wrist=wpositive, fatherId=frmaster[2]}
  [373] = {x=-15.454983, y=28.224383, z=96.64176, rx=-178.000236, ry=-0.000067, rz=-0.000751, shoulder=lefty, elbow=epositive, wrist=wpositive, fatherId=frmaster[2]}
  [374] = {x=-16.453358, y=28.224119, z=96.643571, rx=-178.000024, ry=-0.000343, rz=0.000025, shoulder=lefty, elbow=epositive, wrist=wpositive, fatherId=frmaster[2]}
  [375] = {x=-17.450206, y=28.226407, z=96.645317, rx=-177.999631, ry=0.000277, rz=0.000216, shoulder=lefty, elbow=epositive, wrist=wpositive, fatherId=frmaster[2]}
  [376] = {x=-18.447036, y=28.227318, z=96.643391, rx=-177.999403, ry=0.00001, rz=-0.000016, shoulder=lefty, elbow=epositive, wrist=wpositive, fatherId=frmaster[2]}
  [377] = {x=-19.450839, y=28.225008, z=96.646257, rx=-178.000155, ry=-0.000027, rz=0.000733, shoulder=lefty, elbow=epositive, wrist=wpositive, fatherId=frmaster[2]}
  [378] = {x=-20.445634, y=28.224696, z=96.64544, rx=-177.999908, ry=-0.00028, rz=0.000478, shoulder=lefty, elbow=epositive, wrist=wpositive, fatherId=frmaster[2]}
  [379] = {x=-21.440005, y=28.226695, z=96.644559, rx=-177.999651, ry=-0.000529, rz=-0.000781, shoulder=lefty, elbow=epositive, wrist=wpositive, fatherId=frmaster[2]}
  [380] = {x=-22.440366, y=28.225762, z=96.640108, rx=-177.99923, ry=0.000154, rz=0.000376, shoulder=lefty, elbow=epositive, wrist=wpositive, fatherId=frmaster[2]}
  [381] = {x=-23.432527, y=28.22527, z=96.640306, rx=-177.99994, ry=0.000098, rz=0.000094, shoulder=lefty, elbow=epositive, wrist=wpositive, fatherId=frmaster[2]}
  [382] = {x=-24.432638, y=28.226384, z=96.640553, rx=-177.999665, ry=-0.000098, rz=-0.000192, shoulder=lefty, elbow=epositive, wrist=wpositive, fatherId=frmaster[2]}
  [383] = {x=-25.43162, y=28.226218, z=96.645518, rx=-178.000364, ry=-0.000109, rz=-0.000497, shoulder=lefty, elbow=epositive, wrist=wpositive, fatherId=frmaster[2]}
  [384] = {x=-26.429866, y=28.226107, z=96.63854, rx=-177.999087, ry=-0.000469, rz=0.000208, shoulder=lefty, elbow=epositive, wrist=wpositive, fatherId=frmaster[2]}
  [385] = {x=-27.426718, y=28.223414, z=96.644594, rx=-178.000753, ry=-0.000299, rz=-0.000119, shoulder=lefty, elbow=epositive, wrist=wpositive, fatherId=frmaster[2]}
  [386] = {x=-28.422568, y=28.225682, z=96.642332, rx=-177.999304, ry=0.000252, rz=-0.000012, shoulder=lefty, elbow=epositive, wrist=wpositive, fatherId=frmaster[2]}
  [387] = {x=-29.418216, y=28.225235, z=96.644744, rx=-177.99997, ry=0.000257, rz=-0.000347, shoulder=lefty, elbow=epositive, wrist=wpositive, fatherId=frmaster[2]}
  [388] = {x=-30.413541, y=28.227147, z=96.638763, rx=-177.999643, ry=0.000092, rz=-0.000671, shoulder=lefty, elbow=epositive, wrist=wpositive, fatherId=frmaster[2]}
  [389] = {x=-31.415484, y=28.22353, z=96.64239, rx=-178.0003, ry=0.000141, rz=-0.000028, shoulder=lefty, elbow=epositive, wrist=wpositive, fatherId=frmaster[2]}
  [390] = {x=-32.409078, y=28.225169, z=96.645935, rx=-177.999952, ry=-0.000003, rz=-0.000388, shoulder=lefty, elbow=epositive, wrist=wpositive, fatherId=frmaster[2]}
  [391] = {x=-33.41031, y=28.226213, z=96.641127, rx=-177.999606, ry=-0.000115, rz=0.000262, shoulder=lefty, elbow=epositive, wrist=wpositive, fatherId=frmaster[2]}
  [392] = {x=-34.41005, y=28.223488, z=96.645854, rx=-178.000237, ry=-0.000053, rz=0.00088, shoulder=lefty, elbow=epositive, wrist=wpositive, fatherId=frmaster[2]}
  [393] = {x=-35.401334, y=28.224817, z=96.642142, rx=-177.999863, ry=-0.000184, rz=-0.000491, shoulder=lefty, elbow=epositive, wrist=wpositive, fatherId=frmaster[2]}
  [394] = {x=-36.399752, y=28.223073, z=96.643221, rx=-178.000477, ry=-0.000118, rz=0.00012, shoulder=lefty, elbow=epositive, wrist=wpositive, fatherId=frmaster[2]}
  [395] = {x=-37.39797, y=28.22481, z=96.644293, rx=-178.000094, ry=-0.000201, rz=-0.000272, shoulder=lefty, elbow=epositive, wrist=wpositive, fatherId=frmaster[2]}
  [396] = {x=-38.395265, y=28.225244, z=96.641776, rx=-177.999703, ry=-0.000279, rz=0.000331, shoulder=lefty, elbow=epositive, wrist=wpositive, fatherId=frmaster[2]}
  [397] = {x=-39.391572, y=28.224288, z=96.643979, rx=-178.000291, ry=-0.000199, rz=-0.000082, shoulder=lefty, elbow=epositive, wrist=wpositive, fatherId=frmaster[2]}
  [398] = {x=-40.387677, y=28.226798, z=96.646178, rx=-177.999882, ry=-0.000262, rz=-0.000498, shoulder=lefty, elbow=epositive, wrist=wpositive, fatherId=frmaster[2]}
  [399] = {x=-41.390867, y=28.225177, z=96.644823, rx=-178.000462, ry=-0.000145, rz=0.000081, shoulder=lefty, elbow=epositive, wrist=wpositive, fatherId=frmaster[2]}
  [400] = {x=-42.385374, y=28.22624, z=96.63991, rx=-177.999046, ry=-0.000339, rz=-0.000342, shoulder=lefty, elbow=epositive, wrist=wpositive, fatherId=frmaster[2]}
  [401] = {x=-43.378683, y=28.224591, z=96.647967, rx=-178.00059, ry=-0.000099, rz=-0.000796, shoulder=lefty, elbow=epositive, wrist=wpositive, fatherId=frmaster[2]}
  [402] = {x=-44.38003, y=28.22492, z=96.647801, rx=-178.000154, ry=-0.000106, rz=-0.00024, shoulder=lefty, elbow=epositive, wrist=wpositive, fatherId=frmaster[2]}
  [403] = {x=-45.372378, y=28.225438, z=96.644001, rx=-177.999702, ry=-0.000141, rz=-0.000687, shoulder=lefty, elbow=epositive, wrist=wpositive, fatherId=frmaster[2]}
  [404] = {x=-46.372515, y=28.226675, z=96.640234, rx=-177.99925, ry=-0.000136, rz=-0.000137, shoulder=lefty, elbow=epositive, wrist=wpositive, fatherId=frmaster[2]}
  [405] = {x=-47.371196, y=28.222807, z=96.645943, rx=-178.00077, ry=0.000144, rz=0.000383, shoulder=lefty, elbow=epositive, wrist=wpositive, fatherId=frmaster[2]}
  [406] = {x=-48.370309, y=28.226154, z=96.638625, rx=-177.99931, ry=0.000028, rz=-0.000074, shoulder=lefty, elbow=epositive, wrist=wpositive, fatherId=frmaster[2]}
  [407] = {x=-49.367994, y=28.224374, z=96.640782, rx=-177.999823, ry=0.000183, rz=0.00044, shoulder=lefty, elbow=epositive, wrist=wpositive, fatherId=frmaster[2]}
  [408] = {x=-50.365486, y=28.226041, z=96.642946, rx=-177.999336, ry=0.000217, rz=0.000951, shoulder=lefty, elbow=epositive, wrist=wpositive, fatherId=frmaster[2]}
  [409] = {x=-51.362041, y=28.225113, z=96.641518, rx=-177.999834, ry=0.000378, rz=0.000459, shoulder=lefty, elbow=epositive, wrist=wpositive, fatherId=frmaster[2]}
  [410] = {x=-52.358988, y=28.223796, z=96.644845, rx=-178.00043, ry=-0.000349, rz=-0.000482, shoulder=lefty, elbow=epositive, wrist=wpositive, fatherId=frmaster[2]}
  [411] = {x=-53.354587, y=28.22491, z=96.639885, rx=-177.999917, ry=-0.000303, rz=0.00002, shoulder=lefty, elbow=epositive, wrist=wpositive, fatherId=frmaster[2]}
  [412] = {x=-54.349494, y=28.225753, z=96.639686, rx=-177.999396, ry=-0.000246, rz=-0.000494, shoulder=lefty, elbow=epositive, wrist=wpositive, fatherId=frmaster[2]}
  [413] = {x=-55.351731, y=28.223756, z=96.644274, rx=-177.999867, ry=-0.00003, rz=-0.000024, shoulder=lefty, elbow=epositive, wrist=wpositive, fatherId=frmaster[2]}
  [414] = {x=-56.345571, y=28.225406, z=96.64051, rx=-177.999329, ry=0.000037, rz=0.000456, shoulder=lefty, elbow=epositive, wrist=wpositive, fatherId=frmaster[2]}
  [415] = {x=-57.346761, y=28.224237, z=96.641534, rx=-177.999785, ry=0.000257, rz=0.00092, shoulder=lefty, elbow=epositive, wrist=wpositive, fatherId=frmaster[2]}
  [416] = {x=-58.339147, y=28.224095, z=96.647247, rx=-178.000224, ry=0.000452, rz=0.00037, shoulder=lefty, elbow=epositive, wrist=wpositive, fatherId=frmaster[2]}
  [417] = {x=-59.340541, y=28.22483, z=96.644752, rx=-177.999765, ry=-0.000325, rz=0.000394, shoulder=lefty, elbow=epositive, wrist=wpositive, fatherId=frmaster[2]}
  [418] = {x=-60.331922, y=28.225449, z=96.646911, rx=-178.000186, ry=-0.000126, rz=-0.000162, shoulder=lefty, elbow=epositive, wrist=wpositive, fatherId=frmaster[2]}
  [419] = {x=-61.33078, y=28.223365, z=96.645616, rx=-178.000609, ry=0.000109, rz=0.00028, shoulder=lefty, elbow=epositive, wrist=wpositive, fatherId=frmaster[2]}
  [420] = {x=-62.329458, y=28.224709, z=96.644341, rx=-178.00003, ry=0.000246, rz=-0.000282, shoulder=lefty, elbow=epositive, wrist=wpositive, fatherId=frmaster[2]}
  [421] = {x=-63.3274, y=28.224537, z=96.647782, rx=-178.000437, ry=0.000492, rz=0.000142, shoulder=lefty, elbow=epositive, wrist=wpositive, fatherId=frmaster[2]}
  [422] = {x=-64.325795, y=28.222817, z=96.647704, rx=-178.000921, ry=-0.000157, rz=0.000127, shoulder=lefty, elbow=epositive, wrist=wpositive, fatherId=frmaster[2]}
  [423] = {x=-65.322919, y=28.224618, z=96.64765, rx=-178.000316, rz=0.000545, shoulder=lefty, elbow=epositive, wrist=wpositive, fatherId=frmaster[2]}
  [424] = {x=-66.319416, y=28.224962, z=96.644088, rx=-177.999703, ry=0.000162, rz=-0.000038, shoulder=lefty, elbow=epositive, wrist=wpositive, fatherId=frmaster[2]}
  [425] = {x=-67.315229, y=28.223763, z=96.645244, rx=-178.000077, ry=0.000424, rz=0.000364, shoulder=lefty, elbow=epositive, wrist=wpositive, fatherId=frmaster[2]}
  [426] = {x=-66.326841, y=28.216418, z=96.645409, rx=-178.000707, ry=0.000292, rz=-0.000051, shoulder=lefty, elbow=epositive, wrist=wpositive, fatherId=frmaster[2]}
  [427] = {x=-65.337928, y=28.2088, z=96.642105, rx=-178.000333, ry=0.000073, rz=0.000532, shoulder=lefty, elbow=epositive, wrist=wpositive, fatherId=frmaster[2]}
  [428] = {x=-64.34882, y=28.204564, z=96.638818, rx=-177.998956, ry=-0.000239, rz=0.000113, shoulder=lefty, elbow=epositive, wrist=wpositive, fatherId=frmaster[2]}
  [429] = {x=-63.358443, y=28.19383, z=96.644944, rx=-178.000556, ry=-0.000251, rz=-0.000333, shoulder=lefty, elbow=epositive, wrist=wpositive, fatherId=frmaster[2]}
  [430] = {x=-62.36684, y=28.186678, z=96.642859, rx=-178.00007, ry=0.000438, rz=0.000667, shoulder=lefty, elbow=epositive, wrist=wpositive, fatherId=frmaster[2]}
  [431] = {x=-61.37601, y=28.181601, z=96.640744, rx=-177.999664, ry=0.000234, rz=0.000227, shoulder=lefty, elbow=epositive, wrist=wpositive, fatherId=frmaster[2]}
  [432] = {x=-60.384094, y=28.172485, z=96.648131, rx=-178.000243, ry=0.000145, rz=-0.000239, shoulder=lefty, elbow=epositive, wrist=wpositive, fatherId=frmaster[2]}
  [433] = {x=-59.399946, y=28.163149, z=96.647277, rx=-178.000823, ry=0.000091, rz=0.000303, shoulder=lefty, elbow=epositive, wrist=wpositive, fatherId=frmaster[2]}
  [434] = {x=-58.407439, y=28.158482, z=96.646368, rx=-178.000393, ry=-0.000099, rz=-0.000157, shoulder=lefty, elbow=epositive, wrist=wpositive, fatherId=frmaster[2]}
  [435] = {x=-57.414217, y=28.152378, z=96.641928, rx=-177.999955, ry=-0.000287, rz=-0.000619, shoulder=lefty, elbow=epositive, wrist=wpositive, fatherId=frmaster[2]}
  [436] = {x=-56.428469, y=28.144656, z=96.642313, rx=-177.999517, ry=-0.000434, rz=-0.000098, shoulder=lefty, elbow=epositive, wrist=wpositive, fatherId=frmaster[2]}
  [437] = {x=-55.43265, y=28.136872, z=96.647352, rx=-177.999954, ry=0.000401, rz=-0.000157, shoulder=lefty, elbow=epositive, wrist=wpositive, fatherId=frmaster[2]}
  [438] = {x=-54.445806, y=28.129897, z=96.644168, rx=-177.999499, ry=0.000259, rz=0.000358, shoulder=lefty, elbow=epositive, wrist=wpositive, fatherId=frmaster[2]}
  [439] = {x=-53.458119, y=28.121407, z=96.645701, rx=-178.000029, ry=0.000241, rz=-0.000142, shoulder=lefty, elbow=epositive, wrist=wpositive, fatherId=frmaster[2]}
  [440] = {x=-52.46965, y=28.111487, z=96.643689, rx=-178.00055, ry=0.000229, rz=0.000355, shoulder=lefty, elbow=epositive, wrist=wpositive, fatherId=frmaster[2]}
  [441] = {x=-51.472812, y=28.106391, z=96.641614, rx=-178.000062, ry=0.000068, rz=-0.00015, shoulder=lefty, elbow=epositive, wrist=wpositive, fatherId=frmaster[2]}
  [442] = {x=-50.483251, y=28.098406, z=96.644324, rx=-178.000566, ry=0.00007, rz=-0.000672, shoulder=lefty, elbow=epositive, wrist=wpositive, fatherId=frmaster[2]}
  [443] = {x=-49.49356, y=28.093914, z=96.63877, rx=-177.999079, ry=-0.000177, rz=-0.000184, shoulder=lefty, elbow=epositive, wrist=wpositive, fatherId=frmaster[2]}
  [444] = {x=-48.510597, y=28.082794, z=96.642755, rx=-177.999574, ry=-0.000128, rz=0.000274, shoulder=lefty, elbow=epositive, wrist=wpositive, fatherId=frmaster[2]}
  [445] = {x=-47.518947, y=28.074133, z=96.646593, rx=-178.001045, ry=0.000022, rz=-0.00027, shoulder=lefty, elbow=epositive, wrist=wpositive, fatherId=frmaster[2]}
  [446] = {x=-46.52732, y=28.07019, z=96.642197, rx=-177.999533, ry=-0.000218, rz=0.000195, shoulder=lefty, elbow=epositive, wrist=wpositive, fatherId=frmaster[2]}
  [447] = {x=-45.534612, y=28.063585, z=96.642476, rx=-177.999996, ry=-0.000188, rz=-0.000356, shoulder=lefty, elbow=epositive, wrist=wpositive, fatherId=frmaster[2]}
  [448] = {x=-44.549362, y=28.055289, z=96.639295, rx=-177.999468, ry=-0.000254, rz=0.00009, shoulder=lefty, elbow=epositive, wrist=wpositive, fatherId=frmaster[2]}
  [449] = {x=-43.555006, y=28.047082, z=96.640762, rx=-177.999913, ry=-0.000209, rz=-0.000481, shoulder=lefty, elbow=epositive, wrist=wpositive, fatherId=frmaster[2]}
  [450] = {x=-42.568585, y=28.040759, z=96.642299, rx=-177.999367, ry=-0.000265, rz=-0.000056, shoulder=lefty, elbow=epositive, wrist=wpositive, fatherId=frmaster[2]}
  [451] = {x=-41.581109, y=28.031854, z=96.640214, rx=-177.999804, ry=-0.000178, rz=0.000366, shoulder=lefty, elbow=epositive, wrist=wpositive, fatherId=frmaster[2]}
  [452] = {x=-40.584666, y=28.024325, z=96.642822, rx=-178.000223, ry=-0.000114, rz=-0.000228, shoulder=lefty, elbow=epositive, wrist=wpositive, fatherId=frmaster[2]}
  [453] = {x=-39.595981, y=28.017438, z=96.645453, rx=-178.000641, ry=-0.00001, rz=0.000173, shoulder=lefty, elbow=epositive, wrist=wpositive, fatherId=frmaster[2]}
  [454] = {x=-38.606559, y=28.010411, z=96.64454, rx=-178.000062, ry=-0.000049, rz=-0.000429, shoulder=lefty, elbow=epositive, wrist=wpositive, fatherId=frmaster[2]}
  [455] = {x=-37.616127, y=28.001976, z=96.648346, rx=-178.000463, ry=0.000069, rz=-0.000048, shoulder=lefty, elbow=epositive, wrist=wpositive, fatherId=frmaster[2]}
  [456] = {x=-36.625373, y=27.995861, z=96.643789, rx=-177.999867, ry=0.000035, rz=-0.000658, shoulder=lefty, elbow=epositive, wrist=wpositive, fatherId=frmaster[2]}
  [457] = {x=-35.633592, y=27.988353, z=96.64395, rx=-178.00025, ry=0.000162, rz=-0.000284, shoulder=lefty, elbow=epositive, wrist=wpositive, fatherId=frmaster[2]}
  [458] = {x=-34.649112, y=27.978964, z=96.648941, rx=-178.000633, ry=0.000333, rz=0.000071, shoulder=lefty, elbow=epositive, wrist=wpositive, fatherId=frmaster[2]}
  [459] = {x=-33.65615, y=27.973604, z=96.645489, rx=-178.000011, ry=0.000312, rz=0.000437, shoulder=lefty, elbow=epositive, wrist=wpositive, fatherId=frmaster[2]}
  [460] = {x=-32.670288, y=27.965138, z=96.646823, rx=-178.000376, ry=0.000492, rz=0.000784, shoulder=lefty, elbow=epositive, wrist=wpositive, fatherId=frmaster[2]}
  [461] = {x=-31.676571, y=27.958148, z=96.644512, rx=-177.999882, ry=-0.000412, rz=-0.000295, shoulder=lefty, elbow=epositive, wrist=wpositive, fatherId=frmaster[2]}
  [462] = {x=-30.689303, y=27.950634, z=96.642175, rx=-178.000232, ry=-0.000225, rz=0.000045, shoulder=lefty, elbow=epositive, wrist=wpositive, fatherId=frmaster[2]}
  [463] = {x=-29.70135, y=27.944162, z=96.644643, rx=-177.999585, ry=-0.000191, rz=0.000368, shoulder=lefty, elbow=epositive, wrist=wpositive, fatherId=frmaster[2]}
  [464] = {x=-28.704029, y=27.937016, z=96.643378, rx=-177.999907, ry=-0.000023, rz=-0.000313, shoulder=lefty, elbow=epositive, wrist=wpositive, fatherId=frmaster[2]}
  [465] = {x=-27.713957, y=27.927938, z=96.646943, rx=-178.000227, ry=0.000191, rz=-0.000013, shoulder=lefty, elbow=epositive, wrist=wpositive, fatherId=frmaster[2]}
  [466] = {x=-26.723539, y=27.921209, z=96.642097, rx=-177.999555, ry=0.000231, rz=-0.000703, shoulder=lefty, elbow=epositive, wrist=wpositive, fatherId=frmaster[2]}
  [467] = {x=-25.74186, y=27.914632, z=96.645605, rx=-178.000023, ry=-0.000407, rz=0.000167, shoulder=lefty, elbow=epositive, wrist=wpositive, fatherId=frmaster[2]}
  [468] = {x=-24.749484, y=27.906521, z=96.641881, rx=-177.999334, ry=-0.000356, rz=0.000456, shoulder=lefty, elbow=epositive, wrist=wpositive, fatherId=frmaster[2]}
  [469] = {x=-23.756373, y=27.899434, z=96.646413, rx=-178.000604, ry=0.000056, rz=-0.000274, shoulder=lefty, elbow=epositive, wrist=wpositive, fatherId=frmaster[2]}
  [470] = {x=-22.770785, y=27.891616, z=96.647455, rx=-177.999905, ry=0.000152, rz=0.000991, shoulder=lefty, elbow=epositive, wrist=wpositive, fatherId=frmaster[2]}
  [471] = {x=-21.775746, y=27.883288, z=96.644735, rx=-178.000173, ry=0.000397, rz=0.000252, shoulder=lefty, elbow=epositive, wrist=wpositive, fatherId=frmaster[2]}
  [472] = {x=-20.789732, y=27.876327, z=96.642049, rx=-177.999623, ry=-0.000395, rz=0.00009, shoulder=lefty, elbow=epositive, wrist=wpositive, fatherId=frmaster[2]}
  [473] = {x=-19.801454, y=27.868274, z=96.644091, rx=-177.999881, ry=-0.000103, rz=0.000328, shoulder=lefty, elbow=epositive, wrist=wpositive, fatherId=frmaster[2]}
  [474] = {x=-18.803915, y=27.860998, z=96.642403, rx=-178.000122, ry=0.00016, rz=-0.000438, shoulder=lefty, elbow=epositive, wrist=wpositive, fatherId=frmaster[2]}
  [475] = {x=-17.814314, y=27.855258, z=96.640752, rx=-177.99938, ry=0.000273, rz=-0.000208, shoulder=lefty, elbow=epositive, wrist=wpositive, fatherId=frmaster[2]}
  [476] = {x=-16.824605, y=27.848048, z=96.643817, rx=-177.999783, ry=-0.000308, rz=-0.000416, shoulder=lefty, elbow=epositive, wrist=wpositive, fatherId=frmaster[2]}
  [477] = {x=-15.840837, y=27.837837, z=96.643285, rx=-178.000014, ry=0.000041, rz=0.00079, shoulder=lefty, elbow=epositive, wrist=wpositive, fatherId=frmaster[2]}
  [478] = {x=-14.848458, y=27.831971, z=96.642609, rx=-178.000227, ry=0.000361, rz=-0.000009, shoulder=lefty, elbow=epositive, wrist=wpositive, fatherId=frmaster[2]}
  [479] = {x=-13.856267, y=27.825931, z=96.638284, rx=-177.999629, ry=-0.000403, rz=-0.000227, shoulder=lefty, elbow=epositive, wrist=wpositive, fatherId=frmaster[2]}
  [480] = {x=-12.869825, y=27.816739, z=96.647169, rx=-178.000811, ry=0.00017, rz=-0.000065, shoulder=lefty, elbow=epositive, wrist=wpositive, fatherId=frmaster[2]}
  [481] = {x=-11.874392, y=27.80976, z=96.643926, rx=-178.000016, ry=0.00031, rz=0.000108, shoulder=lefty, elbow=epositive, wrist=wpositive, fatherId=frmaster[2]}
  [482] = {x=-10.887747, y=27.802791, z=96.64066, rx=-177.999406, ry=-0.000408, rz=-0.000138, shoulder=lefty, elbow=epositive, wrist=wpositive, fatherId=frmaster[2]}
  [483] = {x=-9.898755, y=27.794836, z=96.642124, rx=-177.999582, ry=-0.000022, rz=0.00001, shoulder=lefty, elbow=epositive, wrist=wpositive, fatherId=frmaster[2]}
  [484] = {x=-8.908494, y=27.785688, z=96.648315, rx=-178.000725, ry=0.000581, rz=0.000138, shoulder=lefty, elbow=epositive, wrist=wpositive, fatherId=frmaster[2]}
  [485] = {x=-7.919194, y=27.779918, z=96.646028, rx=-178.000093, ry=-0.000122, rz=-0.000136, shoulder=lefty, elbow=epositive, wrist=wpositive, fatherId=frmaster[2]}
  [486] = {x=-6.927613, y=27.773275, z=96.640032, rx=-177.999264, ry=0.000066, rz=-0.000001, shoulder=lefty, elbow=epositive, wrist=wpositive, fatherId=frmaster[2]}
  [487] = {x=-5.935743, y=27.76517, z=96.647193, rx=-178.000572, ry=-0.000198, rz=-0.000314, shoulder=lefty, elbow=epositive, wrist=wpositive, fatherId=frmaster[2]}
  [488] = {x=-4.950822, y=27.758703, z=96.645943, rx=-177.999733, ry=0.000036, rz=0.000795, shoulder=lefty, elbow=epositive, wrist=wpositive, fatherId=frmaster[2]}
  [489] = {x=-3.957353, y=27.751947, z=96.640847, rx=-178.000051, ry=-0.000439, rz=-0.00051, shoulder=lefty, elbow=epositive, wrist=wpositive, fatherId=frmaster[2]}
  [490] = {x=-2.97017, y=27.744433, z=96.640633, rx=-177.999195, ry=-0.000195, rz=0.000574, shoulder=lefty, elbow=epositive, wrist=wpositive, fatherId=frmaster[2]}
  [491] = {x=-1.973239, y=27.736868, z=96.645036, rx=-178.000271, ry=0.000461, rz=-0.000363, shoulder=lefty, elbow=epositive, wrist=wpositive, fatherId=frmaster[2]}
  [492] = {x=-0.985437, y=27.730424, z=96.640983, rx=-177.999599, ry=-0.000182, rz=-0.000697, shoulder=lefty, elbow=epositive, wrist=wpositive, fatherId=frmaster[2]}
  [493] = {x=0.004785, y=27.723108, z=96.641663, rx=-177.99969, ry=0.000297, rz=0.000356, shoulder=lefty, elbow=epositive, wrist=wpositive, fatherId=frmaster[2]}
  [494] = {x=0.988125, y=27.707666, z=96.639905, rx=-177.99901, ry=-0.000296, rz=-0.00002, shoulder=lefty, elbow=epositive, wrist=wpositive, fatherId=frmaster[2]}
  [495] = {x=1.982359, y=27.692532, z=96.642767, rx=-178.000054, ry=0.00043, rz=-0.000009, shoulder=lefty, elbow=epositive, wrist=wpositive, fatherId=frmaster[2]}
  [496] = {x=2.975729, y=27.680756, z=96.645561, rx=-178.000324, ry=0.000045, rz=-0.00041, shoulder=lefty, elbow=epositive, wrist=wpositive, fatherId=frmaster[2]}
  [497] = {x=3.962233, y=27.665619, z=96.644658, rx=-178.000596, ry=-0.000303, rz=0.000185, shoulder=lefty, elbow=epositive, wrist=wpositive, fatherId=frmaster[2]}
  [498] = {x=4.950932, y=27.650868, z=96.648528, rx=-178.000647, ry=0.00025, rz=0.000164, shoulder=lefty, elbow=epositive, wrist=wpositive, fatherId=frmaster[2]}
  [499] = {x=5.938953, y=27.638335, z=96.643783, rx=-177.999932, ry=-0.000324, rz=-0.00025, shoulder=lefty, elbow=epositive, wrist=wpositive, fatherId=frmaster[2]}
  [500] = {x=6.92946, y=27.625027, z=96.643767, rx=-177.999965, ry=0.000235, rz=0.000718, shoulder=lefty, elbow=epositive, wrist=wpositive, fatherId=frmaster[2]}
  [501] = {x=7.919911, y=27.611689, z=96.639994, rx=-177.999235, ry=-0.000329, rz=0.000278, shoulder=lefty, elbow=epositive, wrist=wpositive, fatherId=frmaster[2]}
  [502] = {x=8.913246, y=27.596362, z=96.649429, rx=-178.001188, ry=0.00073, rz=0.000202, shoulder=lefty, elbow=epositive, wrist=wpositive, fatherId=frmaster[2]}
  [503] = {x=9.905233, y=27.585719, z=96.641787, rx=-177.999474, ry=-0.000071, rz=-0.000247, shoulder=lefty, elbow=epositive, wrist=wpositive, fatherId=frmaster[2]}
  [504] = {x=10.890866, y=27.570341, z=96.647417, rx=-178.000669, ry=-0.000095, rz=0.000266, shoulder=lefty, elbow=epositive, wrist=wpositive, fatherId=frmaster[2]}
  [505] = {x=11.878543, y=27.555558, z=96.640762, rx=-177.999695, ry=0.000278, rz=0.00019, shoulder=lefty, elbow=epositive, wrist=wpositive, fatherId=frmaster[2]}
  [506] = {x=12.873885, y=27.545412, z=96.642444, rx=-177.999897, ry=-0.000017, rz=-0.000306, shoulder=lefty, elbow=epositive, wrist=wpositive, fatherId=frmaster[2]}
  [507] = {x=13.863061, y=27.529609, z=96.645265, rx=-178.000099, ry=-0.000267, rz=-0.000825, shoulder=lefty, elbow=epositive, wrist=wpositive, fatherId=frmaster[2]}
  [508] = {x=14.853826, y=27.516551, z=96.647976, rx=-178.000063, ry=0.000376, rz=0.000049, shoulder=lefty, elbow=epositive, wrist=wpositive, fatherId=frmaster[2]}
  [509] = {x=15.844873, y=27.502341, z=96.646853, rx=-178.00025, ry=0.000133, rz=-0.000479, shoulder=lefty, elbow=epositive, wrist=wpositive, fatherId=frmaster[2]}
  [510] = {x=16.828259, y=27.488003, z=96.64567, rx=-178.000439, ry=-0.000072, rz=-0.000013, shoulder=lefty, elbow=epositive, wrist=wpositive, fatherId=frmaster[2]}
  [511] = {x=17.82087, y=27.476588, z=96.640621, rx=-177.999647, ry=-0.000564, rz=-0.000551, shoulder=lefty, elbow=epositive, wrist=wpositive, fatherId=frmaster[2]}
  [512] = {x=18.807872, y=27.461929, z=96.640373, rx=-177.999583, ry=0.000132, rz=0.000283, shoulder=lefty, elbow=epositive, wrist=wpositive, fatherId=frmaster[2]}
  [513] = {x=19.803115, y=27.449911, z=96.644816, rx=-177.999737, ry=-0.000083, rz=-0.000299, shoulder=lefty, elbow=epositive, wrist=wpositive, fatherId=frmaster[2]}
  [514] = {x=20.791589, y=27.434424, z=96.645476, rx=-177.999894, ry=-0.000261, rz=0.000113, shoulder=lefty, elbow=epositive, wrist=wpositive, fatherId=frmaster[2]}
  [515] = {x=21.780564, y=27.421433, z=96.646003, rx=-178.000044, ry=-0.000436, rz=-0.00048, shoulder=lefty, elbow=epositive, wrist=wpositive, fatherId=frmaster[2]}
  [516] = {x=22.772025, y=27.407941, z=96.642677, rx=-177.999942, ry=0.000281, rz=0.000314, shoulder=lefty, elbow=epositive, wrist=wpositive, fatherId=frmaster[2]}
  [517] = {x=23.763577, y=27.394483, z=96.644106, rx=-178.000074, ry=0.000121, rz=-0.000306, shoulder=lefty, elbow=epositive, wrist=wpositive, fatherId=frmaster[2]}
  [518] = {x=24.748377, y=27.377517, z=96.641727, rx=-178.000208, ry=-0.000002, rz=0.000068, shoulder=lefty, elbow=epositive, wrist=wpositive, fatherId=frmaster[2]}
  [519] = {x=25.741513, y=27.366989, z=96.639178, rx=-177.999364, ry=-0.000427, rz=-0.000563, shoulder=lefty, elbow=epositive, wrist=wpositive, fatherId=frmaster[2]}
  [520] = {x=26.727989, y=27.352881, z=96.641425, rx=-177.999483, ry=-0.000538, rz=-0.000217, shoulder=lefty, elbow=epositive, wrist=wpositive, fatherId=frmaster[2]}
  [521] = {x=27.716974, y=27.33833, z=96.639792, rx=-177.999341, ry=0.000241, rz=0.000512, shoulder=lefty, elbow=epositive, wrist=wpositive, fatherId=frmaster[2]}
  [522] = {x=28.706062, y=27.323849, z=96.642917, rx=-177.999441, ry=0.000144, rz=0.000829, shoulder=lefty, elbow=epositive, wrist=wpositive, fatherId=frmaster[2]}
  [523] = {x=29.695984, y=27.310737, z=96.645859, rx=-178.000495, ry=0.000329, rz=0.000142, shoulder=lefty, elbow=epositive, wrist=wpositive, fatherId=frmaster[2]}
  [524] = {x=30.687698, y=27.295951, z=96.649858, rx=-178.000579, ry=0.000248, rz=0.000431, shoulder=lefty, elbow=epositive, wrist=wpositive, fatherId=frmaster[2]}
  [525] = {x=31.680162, y=27.282624, z=96.645021, rx=-178.000658, ry=0.000162, rz=-0.000267, shoulder=lefty, elbow=epositive, wrist=wpositive, fatherId=frmaster[2]}
  [526] = {x=32.67382, y=27.269739, z=96.644951, rx=-178.000728, ry=0.000088, rz=-0.000989, shoulder=lefty, elbow=epositive, wrist=wpositive, fatherId=frmaster[2]}
  [527] = {x=33.659451, y=27.257708, z=96.644835, rx=-177.999841, ry=-0.000237, rz=0.000284, shoulder=lefty, elbow=epositive, wrist=wpositive, fatherId=frmaster[2]}
  [528] = {x=34.647938, y=27.240543, z=96.645634, rx=-178.000861, ry=0.000022, rz=0.000533, shoulder=lefty, elbow=epositive, wrist=wpositive, fatherId=frmaster[2]}
  [529] = {x=35.636566, y=27.227125, z=96.646317, rx=-178.000915, ry=-0.000003, rz=-0.000223, shoulder=lefty, elbow=epositive, wrist=wpositive, fatherId=frmaster[2]}
  [530] = {x=36.626297, y=27.214239, z=96.643097, rx=-178.000006, ry=-0.000316, rz=0.000015, shoulder=lefty, elbow=epositive, wrist=wpositive, fatherId=frmaster[2]}
  [531] = {x=37.617583, y=27.200676, z=96.644606, rx=-178.000045, ry=-0.000329, rz=0.00023, shoulder=lefty, elbow=epositive, wrist=wpositive, fatherId=frmaster[2]}
  [532] = {x=38.609352, y=27.189718, z=96.645954, rx=-178.000076, ry=-0.000339, rz=-0.000561, shoulder=lefty, elbow=epositive, wrist=wpositive, fatherId=frmaster[2]}
  [533] = {x=39.5955, y=27.171913, z=96.648308, rx=-178.001061, ry=-0.000008, rz=0.000624, shoulder=lefty, elbow=epositive, wrist=wpositive, fatherId=frmaster[2]}
  [534] = {x=40.589848, y=27.160957, z=96.64177, rx=-178.000123, ry=-0.000309, rz=-0.000178, shoulder=lefty, elbow=epositive, wrist=wpositive, fatherId=frmaster[2]}
  [535] = {x=41.577592, y=27.146353, z=96.640024, rx=-178.000139, ry=-0.00027, rz=-0.000005, shoulder=lefty, elbow=epositive, wrist=wpositive, fatherId=frmaster[2]}
  [536] = {x=42.566539, y=27.132291, z=96.643051, rx=-178.000145, ry=-0.00022, rz=0.000144, shoulder=lefty, elbow=epositive, wrist=wpositive, fatherId=frmaster[2]}
  [537] = {x=43.556969, y=27.117689, z=96.642095, rx=-178.000143, ry=-0.000167, rz=0.000288, shoulder=lefty, elbow=epositive, wrist=wpositive, fatherId=frmaster[2]}
  [538] = {x=44.547872, y=27.10573, z=96.640964, rx=-178.000135, ry=-0.000112, rz=0.000425, shoulder=lefty, elbow=epositive, wrist=wpositive, fatherId=frmaster[2]}
  [539] = {x=45.539977, y=27.094362, z=96.644608, rx=-178.000116, ry=-0.000047, rz=-0.000461, shoulder=lefty, elbow=epositive, wrist=wpositive, fatherId=frmaster[2]}
  [540] = {x=46.525396, y=27.079377, z=96.644321, rx=-178.000099, ry=0.000055, rz=0.000645, shoulder=lefty, elbow=epositive, wrist=wpositive, fatherId=frmaster[2]}
  [541] = {x=47.520097, y=27.06819, z=96.639997, rx=-177.999115, ry=-0.000186, rz=-0.000253, shoulder=lefty, elbow=epositive, wrist=wpositive, fatherId=frmaster[2]}
  [542] = {x=48.508211, y=27.053334, z=96.640469, rx=-177.999081, ry=-0.000074, rz=-0.000177, shoulder=lefty, elbow=epositive, wrist=wpositive, fatherId=frmaster[2]}
  [543] = {x=49.497913, y=27.037956, z=96.645677, rx=-177.999986, ry=0.000363, rz=-0.000127, shoulder=lefty, elbow=epositive, wrist=wpositive, fatherId=frmaster[2]}
  [544] = {x=50.486909, y=27.024961, z=96.641929, rx=-178.000231, ry=-0.000399, rz=-0.000431, shoulder=lefty, elbow=epositive, wrist=wpositive, fatherId=frmaster[2]}
  [545] = {x=51.479318, y=27.009813, z=96.64789, rx=-178.001118, ry=0.000055, rz=-0.00041, shoulder=lefty, elbow=epositive, wrist=wpositive, fatherId=frmaster[2]}
  [546] = {x=52.471703, y=26.998593, z=96.64493, rx=-178.000105, ry=-0.000132, rz=-0.000377, shoulder=lefty, elbow=epositive, wrist=wpositive, fatherId=frmaster[2]}
  [547] = {x=53.457506, y=26.983677, z=96.64677, rx=-178.000038, ry=0.000043, rz=-0.000369, shoulder=lefty, elbow=epositive, wrist=wpositive, fatherId=frmaster[2]}
  [548] = {x=54.444811, y=26.968357, z=96.644559, rx=-177.999963, ry=0.00022, rz=0.000632, shoulder=lefty, elbow=epositive, wrist=wpositive, fatherId=frmaster[2]}
  [549] = {x=55.441887, y=26.955878, z=96.647014, rx=-178.000816, ry=0.000699, rz=-0.000391, shoulder=lefty, elbow=epositive, wrist=wpositive, fatherId=frmaster[2]}
  [550] = {x=56.429668, y=26.9437, z=96.640565, rx=-178.000085, ry=-0.000326, rz=-0.000765, shoulder=lefty, elbow=epositive, wrist=wpositive, fatherId=frmaster[2]}
  [551] = {x=57.420878, y=26.929501, z=96.643835, rx=-177.999984, ry=-0.000127, rz=-0.00082, shoulder=lefty, elbow=epositive, wrist=wpositive, fatherId=frmaster[2]}
  [552] = {x=58.404351, y=26.914722, z=96.646975, rx=-177.999885, ry=0.000107, rz=0.000118, shoulder=lefty, elbow=epositive, wrist=wpositive, fatherId=frmaster[2]}
  [553] = {x=59.397502, y=26.90295, z=96.645966, rx=-177.999769, ry=0.00031, rz=0.00005, shoulder=lefty, elbow=epositive, wrist=wpositive, fatherId=frmaster[2]}
  [554] = {x=60.38291, y=26.887145, z=96.640916, rx=-177.999965, ry=-0.000331, rz=0.000616, shoulder=lefty, elbow=epositive, wrist=wpositive, fatherId=frmaster[2]}
  [555] = {x=61.378761, y=26.875898, z=96.640585, rx=-177.999833, ry=-0.000116, rz=-0.000484, shoulder=lefty, elbow=epositive, wrist=wpositive, fatherId=frmaster[2]}
  [556] = {x=62.367626, y=26.862101, z=96.645098, rx=-177.999699, ry=0.000141, rz=0.00039, shoulder=lefty, elbow=epositive, wrist=wpositive, fatherId=frmaster[2]}
  [557] = {x=63.356924, y=26.847662, z=96.645491, rx=-177.999874, ry=-0.000479, rz=-0.000099, shoulder=lefty, elbow=epositive, wrist=wpositive, fatherId=frmaster[2]}
  [558] = {x=64.348805, y=26.833378, z=96.641777, rx=-177.999726, ry=-0.000217, rz=-0.000238, shoulder=lefty, elbow=epositive, wrist=wpositive, fatherId=frmaster[2]}
  [559] = {x=65.333019, y=26.818396, z=96.646773, rx=-178.000516, ry=0.00043, rz=0.000596, shoulder=lefty, elbow=epositive, wrist=wpositive, fatherId=frmaster[2]}
  [560] = {x=66.326521, y=26.804392, z=96.643689, rx=-178.000672, ry=-0.000175, rz=0.000071, shoulder=lefty, elbow=epositive, wrist=wpositive, fatherId=frmaster[2]}
  [561] = {x=67.312905, y=26.791279, z=96.640498, rx=-177.999569, ry=-0.000211, rz=0.000893, shoulder=lefty, elbow=epositive, wrist=wpositive, fatherId=frmaster[2]}
  [562] = {x=66.595588, y=27.110878, z=97.57913, rx=-178.205279, ry=0.882749, rz=-0.014528, shoulder=lefty, elbow=epositive, wrist=wpositive, fatherId=frmaster[2]}
  [563] = {x=66.462529, y=27.720789, z=98.013316, rx=-178.580694, ry=1.408727, rz=-0.016888, shoulder=lefty, elbow=epositive, wrist=wpositive, fatherId=frmaster[2]}
  [564] = {x=65.908316, y=27.794061, z=98.182744, rx=-179.024092, ry=1.745725, rz=-0.014778, shoulder=lefty, elbow=epositive, wrist=wpositive, fatherId=frmaster[2]}
  [565] = {x=65.521755, y=28.36304, z=98.101307, rx=-179.761562, ry=1.985468, rz=-0.00446, shoulder=lefty, elbow=epositive, wrist=wpositive, fatherId=frmaster[2]}
  [566] = {x=65.508538, y=28.582756, z=97.995173, rx=-179.999828, ry=1.999842, rz=-0.000584, shoulder=lefty, elbow=epositive, wrist=wpositive, fatherId=frmaster[2]}
  [567] = {x=65.520727, y=28.01913, z=97.992373, rx=-179.999542, ry=1.999973, rz=-0.000328, shoulder=lefty, elbow=epositive, wrist=wpositive, fatherId=frmaster[2]}
  [568] = {x=65.53426, y=27.526652, z=97.998215, rx=179.999867, ry=2.000286, rz=-0.000676, shoulder=lefty, elbow=epositive, wrist=wpositive, fatherId=frmaster[2]}
  [569] = {x=65.559171, y=26.544536, z=97.99127, rx=-179.999446, ry=2.000203, rz=-0.000352, shoulder=lefty, elbow=epositive, wrist=wpositive, fatherId=frmaster[2]}
  [570] = {x=65.583129, y=25.558788, z=97.998034, rx=-179.999993, ry=1.999617, rz=-0.000501, shoulder=lefty, elbow=epositive, wrist=wpositive, fatherId=frmaster[2]}
  [571] = {x=65.606562, y=24.574151, z=97.999737, rx=179.999757, ry=1.999878, rz=-0.000259, shoulder=lefty, elbow=epositive, wrist=wpositive, fatherId=frmaster[2]}
  [572] = {x=65.629083, y=23.58842, z=97.992394, rx=-179.999555, ry=1.999792, rz=-0.000046, shoulder=lefty, elbow=epositive, wrist=wpositive, fatherId=frmaster[2]}
  [573] = {x=65.659081, y=22.605065, z=97.993748, rx=-179.999762, ry=2.000051, rz=-0.000879, shoulder=lefty, elbow=epositive, wrist=wpositive, fatherId=frmaster[2]}
  [574] = {x=65.678882, y=21.620297, z=97.998943, rx=179.999987, ry=2.000307, rz=0.000252, shoulder=lefty, elbow=epositive, wrist=wpositive, fatherId=frmaster[2]}
  [575] = {x=65.704906, y=20.637747, z=97.994922, rx=-179.999586, ry=1.999345, rz=-0.000023, shoulder=lefty, elbow=epositive, wrist=wpositive, fatherId=frmaster[2]}
  [576] = {x=65.731486, y=19.653591, z=97.990765, rx=-179.999801, ry=1.99958, rz=-0.000925, shoulder=lefty, elbow=epositive, wrist=wpositive, fatherId=frmaster[2]}
  [577] = {x=65.748492, y=18.666355, z=97.99546, rx=179.999946, ry=1.999827, rz=0.000095, shoulder=lefty, elbow=epositive, wrist=wpositive, fatherId=frmaster[2]}
  [578] = {x=65.781074, y=17.685422, z=97.990821, rx=-179.999281, ry=1.999729, rz=-0.000915, shoulder=lefty, elbow=epositive, wrist=wpositive, fatherId=frmaster[2]}
  [579] = {x=65.804419, y=16.700425, z=97.995056, rx=-179.999493, ry=1.999969, rz=0.000029, shoulder=lefty, elbow=epositive, wrist=wpositive, fatherId=frmaster[2]}
  [580] = {x=65.827125, y=15.713792, z=97.999098, rx=179.999349, ry=2.000531, rz=-0.00003, shoulder=lefty, elbow=epositive, wrist=wpositive, fatherId=frmaster[2]}
  [581] = {x=65.848275, y=14.727954, z=97.993841, rx=-179.999925, ry=2.000421, rz=0.000848, shoulder=lefty, elbow=epositive, wrist=wpositive, fatherId=frmaster[2]}
  [582] = {x=65.875738, y=13.744867, z=97.997294, rx=179.999601, ry=1.999769, rz=0.000324, shoulder=lefty, elbow=epositive, wrist=wpositive, fatherId=frmaster[2]}
  [583] = {x=65.903086, y=12.761967, z=97.991443, rx=-179.999632, ry=1.999651, rz=0.000129, shoulder=lefty, elbow=epositive, wrist=wpositive, fatherId=frmaster[2]}
  [584] = {x=65.929387, y=11.778903, z=97.994413, rx=-179.999807, ry=1.999866, rz=-0.00011, shoulder=lefty, elbow=epositive, wrist=wpositive, fatherId=frmaster[2]}
  [585] = {x=65.947154, y=10.789427, z=98.002267, rx=179.999033, ry=2.000413, rz=0.000606, shoulder=lefty, elbow=epositive, wrist=wpositive, fatherId=frmaster[2]}
  [586] = {x=65.979451, y=9.809889, z=97.995474, rx=179.999839, ry=2.00028, rz=-0.0007, shoulder=lefty, elbow=epositive, wrist=wpositive, fatherId=frmaster[2]}
  [587] = {x=66.002741, y=8.825303, z=97.993505, rx=-179.999394, ry=2.000153, rz=-0.000084, shoulder=lefty, elbow=epositive, wrist=wpositive, fatherId=frmaster[2]}
  [588] = {x=66.024066, y=7.839454, z=97.991181, rx=-179.999878, ry=1.999457, rz=0.000188, shoulder=lefty, elbow=epositive, wrist=wpositive, fatherId=frmaster[2]}
  [589] = {x=66.045829, y=6.852629, z=97.993644, rx=179.999943, ry=1.999653, rz=0.000725, shoulder=lefty, elbow=epositive, wrist=wpositive, fatherId=frmaster[2]}
  [590] = {x=66.074777, y=5.869747, z=97.995693, rx=179.999806, ry=1.999842, rz=0.000225, shoulder=lefty, elbow=epositive, wrist=wpositive, fatherId=frmaster[2]}
  [591] = {x=66.102371, y=4.887439, z=97.997385, rx=179.999667, ry=2.000022, rz=-0.000312, shoulder=lefty, elbow=epositive, wrist=wpositive, fatherId=frmaster[2]}
  [592] = {x=66.120564, y=3.900708, z=97.994643, rx=-179.999571, ry=1.999872, rz=0.000081, shoulder=lefty, elbow=epositive, wrist=wpositive, fatherId=frmaster[2]}
  [593] = {x=66.146273, y=2.91708, z=97.991441, rx=-179.999716, ry=2.000035, rz=0.00047, shoulder=lefty, elbow=epositive, wrist=wpositive, fatherId=frmaster[2]}
  [594] = {x=66.171153, y=1.932711, z=97.992941, rx=-179.999858, ry=2.000203, rz=0.000782, shoulder=lefty, elbow=epositive, wrist=wpositive, fatherId=frmaster[2]}
  [595] = {x=66.195151, y=0.947743, z=97.999147, rx=-179.999998, ry=2.000373, rz=0.000016, shoulder=lefty, elbow=epositive, wrist=wpositive, fatherId=frmaster[2]}
  [596] = {x=66.225443, y=-0.0341, z=97.995531, rx=179.999596, ry=1.999626, rz=-0.001065, shoulder=lefty, elbow=epositive, wrist=wpositive, fatherId=frmaster[2]}
  [597] = {x=66.247225, y=-1.019386, z=97.996694, rx=179.99945, ry=1.999774, rz=0.000099, shoulder=lefty, elbow=epositive, wrist=wpositive, fatherId=frmaster[2]}
  [598] = {x=66.267892, y=-2.004832, z=97.993192, rx=-179.999751, ry=1.999593, rz=0.000193, shoulder=lefty, elbow=epositive, wrist=wpositive, fatherId=frmaster[2]}
  [599] = {x=66.296564, y=-2.988016, z=97.994276, rx=-179.999855, ry=1.999732, rz=0.000243, shoulder=lefty, elbow=epositive, wrist=wpositive, fatherId=frmaster[2]}
  [600] = {x=66.324526, y=-3.972258, z=98.000021, rx=179.999093, ry=2.000189, rz=-0.000752, shoulder=lefty, elbow=epositive, wrist=wpositive, fatherId=frmaster[2]}
  [601] = {x=66.342516, y=-4.959686, z=98.001102, rx=179.998943, ry=2.000314, rz=0.000184, shoulder=lefty, elbow=epositive, wrist=wpositive, fatherId=frmaster[2]}
  [602] = {x=66.367924, y=-5.943207, z=97.997331, rx=179.999781, ry=2.00011, rz=0.00005, shoulder=lefty, elbow=epositive, wrist=wpositive, fatherId=frmaster[2]}
  [603] = {x=66.392459, y=-6.927333, z=97.998166, rx=179.999671, ry=2.000222, rz=-0.000128, shoulder=lefty, elbow=epositive, wrist=wpositive, fatherId=frmaster[2]}
  [604] = {x=66.415592, y=-7.910713, z=97.994163, rx=-179.999494, ry=2.000004, rz=0.000625, shoulder=lefty, elbow=epositive, wrist=wpositive, fatherId=frmaster[2]}
  [605] = {x=66.447496, y=-8.893542, z=97.999859, rx=179.999492, ry=2.000427, rz=-0.000674, shoulder=lefty, elbow=epositive, wrist=wpositive, fatherId=frmaster[2]}
  [606] = {x=66.469093, y=-9.878752, z=98.00074, rx=179.999378, ry=2.000518, rz=-0.000042, shoulder=lefty, elbow=epositive, wrist=wpositive, fatherId=frmaster[2]}
  [607] = {x=66.490049, y=-10.865308, z=98.001891, rx=179.999264, ry=2.000605, rz=0.000513, shoulder=lefty, elbow=epositive, wrist=wpositive, fatherId=frmaster[2]}
  [608] = {x=66.518208, y=-11.846946, z=97.998003, rx=-179.999861, ry=2.000362, rz=-0.000002, shoulder=lefty, elbow=epositive, wrist=wpositive, fatherId=frmaster[2]}
  [609] = {x=66.546006, y=-12.830698, z=97.994329, rx=-179.999937, ry=2.000428, rz=-0.00056, shoulder=lefty, elbow=epositive, wrist=wpositive, fatherId=frmaster[2]}
  [610] = {x=66.562695, y=-13.817907, z=98.000376, rx=179.999647, ry=1.999587, rz=0.00049, shoulder=lefty, elbow=epositive, wrist=wpositive, fatherId=frmaster[2]}
  [611] = {x=66.587845, y=-14.800392, z=97.991807, rx=-179.999485, ry=1.999313, rz=-0.00021, shoulder=lefty, elbow=epositive, wrist=wpositive, fatherId=frmaster[2]}
  [612] = {x=66.61303, y=-15.785762, z=97.998128, rx=179.99949, ry=1.99968, rz=-0.000002, shoulder=lefty, elbow=epositive, wrist=wpositive, fatherId=frmaster[2]}
  [613] = {x=66.636689, y=-16.770017, z=97.994968, rx=-179.999639, ry=1.999401, rz=0.000103, shoulder=lefty, elbow=epositive, wrist=wpositive, fatherId=frmaster[2]}
  [614] = {x=66.668554, y=-17.751811, z=97.991799, rx=-179.999678, ry=1.999426, rz=-0.000834, shoulder=lefty, elbow=epositive, wrist=wpositive, fatherId=frmaster[2]}
  [615] = {x=66.690774, y=-18.738009, z=97.993952, rx=-179.999758, ry=1.99945, rz=0.000111, shoulder=lefty, elbow=epositive, wrist=wpositive, fatherId=frmaster[2]}
  [616] = {x=66.713192, y=-19.724361, z=97.996158, rx=179.999509, ry=2.00069, rz=0.000268, shoulder=lefty, elbow=epositive, wrist=wpositive, fatherId=frmaster[2]}
  [617] = {x=66.740235, y=-20.704775, z=97.998156, rx=-179.999882, ry=1.999463, rz=-0.000227, shoulder=lefty, elbow=epositive, wrist=wpositive, fatherId=frmaster[2]}
  [618] = {x=66.759955, y=-21.69313, z=98.001072, rx=179.999083, ry=1.999769, rz=0.000482, shoulder=lefty, elbow=epositive, wrist=wpositive, fatherId=frmaster[2]}
  [619] = {x=66.787796, y=-22.675021, z=97.994161, rx=-179.999714, ry=2.00035, rz=0.000334, shoulder=lefty, elbow=epositive, wrist=wpositive, fatherId=frmaster[2]}
  [620] = {x=66.814207, y=-23.659193, z=97.997567, rx=-179.999757, ry=2.000328, rz=-0.000187, shoulder=lefty, elbow=epositive, wrist=wpositive, fatherId=frmaster[2]}
  [621] = {x=66.839635, y=-24.643693, z=97.996358, rx=-179.999805, ry=2.000288, rz=0.000217, shoulder=lefty, elbow=epositive, wrist=wpositive, fatherId=frmaster[2]}
  [622] = {x=66.864066, y=-25.628249, z=98.000198, rx=179.999196, ry=2.00055, rz=0.000537, shoulder=lefty, elbow=epositive, wrist=wpositive, fatherId=frmaster[2]}
  [623] = {x=66.887276, y=-26.612469, z=97.994842, rx=-179.999905, ry=2.000174, rz=-0.000284, shoulder=lefty, elbow=epositive, wrist=wpositive, fatherId=frmaster[2]}
  [624] = {x=66.909698, y=-27.597212, z=97.99972, rx=-179.999955, ry=2.000105, rz=0.00077, shoulder=lefty, elbow=epositive, wrist=wpositive, fatherId=frmaster[2]}
  [625] = {x=66.940537, y=-28.579706, z=97.995223, rx=-179.999967, ry=2.000016, rz=-0.000251, shoulder=lefty, elbow=epositive, wrist=wpositive, fatherId=frmaster[2]}
  [626] = {x=66.939671, y=-27.594677, z=97.991354, rx=-179.999821, ry=2.000118, rz=-0.000272, shoulder=lefty, elbow=epositive, wrist=wpositive, fatherId=frmaster[2]}
  [627] = {x=66.937503, y=-26.608785, z=97.9977, rx=-179.999672, ry=2.000217, rz=0.000549, shoulder=lefty, elbow=epositive, wrist=wpositive, fatherId=frmaster[2]}
  [628] = {x=66.934733, y=-25.624662, z=97.994836, rx=-179.999527, ry=2.000296, rz=0.000295, shoulder=lefty, elbow=epositive, wrist=wpositive, fatherId=frmaster[2]}
  [629] = {x=66.939244, y=-24.638473, z=98.002153, rx=179.999412, ry=1.999766, rz=-0.00032, shoulder=lefty, elbow=epositive, wrist=wpositive, fatherId=frmaster[2]}
  [630] = {x=66.934602, y=-23.655533, z=97.995237, rx=179.999551, ry=1.99982, rz=0.000231, shoulder=lefty, elbow=epositive, wrist=wpositive, fatherId=frmaster[2]}
  [631] = {x=66.93772, y=-22.668461, z=97.993355, rx=179.999734, ry=1.999869, rz=-0.000336, shoulder=lefty, elbow=epositive, wrist=wpositive, fatherId=frmaster[2]}
  [632] = {x=66.939626, y=-21.681038, z=97.996597, rx=179.999918, ry=1.999912, rz=-0.00002, shoulder=lefty, elbow=epositive, wrist=wpositive, fatherId=frmaster[2]}
  [633] = {x=66.940711, y=-20.694687, z=97.995346, rx=-179.999902, ry=1.999941, rz=-0.000779, shoulder=lefty, elbow=epositive, wrist=wpositive, fatherId=frmaster[2]}
  [634] = {x=66.941169, y=-19.709735, z=97.999295, rx=179.999329, ry=2.00028, rz=-0.000622, shoulder=lefty, elbow=epositive, wrist=wpositive, fatherId=frmaster[2]}
  [635] = {x=66.94063, y=-18.725276, z=97.998831, rx=179.999509, ry=2.000294, rz=-0.000574, shoulder=lefty, elbow=epositive, wrist=wpositive, fatherId=frmaster[2]}
  [636] = {x=66.938776, y=-17.740311, z=97.998393, rx=179.999686, ry=2.000297, rz=0.000397, shoulder=lefty, elbow=epositive, wrist=wpositive, fatherId=frmaster[2]}
  [637] = {x=66.935686, y=-16.755071, z=97.998009, rx=179.999861, ry=2.00029, rz=0.000293, shoulder=lefty, elbow=epositive, wrist=wpositive, fatherId=frmaster[2]}
  [638] = {x=66.940357, y=-15.766301, z=97.997636, rx=-179.999922, ry=2.000274, rz=0.000111, shoulder=lefty, elbow=epositive, wrist=wpositive, fatherId=frmaster[2]}
  [639] = {x=66.935833, y=-14.783678, z=97.993123, rx=-179.99975, ry=2.000249, rz=-0.000146, shoulder=lefty, elbow=epositive, wrist=wpositive, fatherId=frmaster[2]}
  [640] = {x=66.939296, y=-13.798038, z=97.998237, rx=179.999519, ry=2.000542, rz=-0.000489, shoulder=lefty, elbow=epositive, wrist=wpositive, fatherId=frmaster[2]}
  [641] = {x=66.940887, y=-12.810483, z=97.998304, rx=179.999732, ry=2.000503, rz=0.0001, shoulder=lefty, elbow=epositive, wrist=wpositive, fatherId=frmaster[2]}
  [642] = {x=66.941504, y=-11.823722, z=97.989072, rx=-179.99911, ry=2.000131, rz=-0.000379, shoulder=lefty, elbow=epositive, wrist=wpositive, fatherId=frmaster[2]}
  [643] = {x=66.941404, y=-10.838039, z=97.989591, rx=-179.998898, ry=2.00008, rz=0.000056, shoulder=lefty, elbow=epositive, wrist=wpositive, fatherId=frmaster[2]}
  [644] = {x=66.941049, y=-9.854801, z=97.999856, rx=179.99942, ry=2.000668, rz=-0.000559, shoulder=lefty, elbow=epositive, wrist=wpositive, fatherId=frmaster[2]}
  [645] = {x=66.938994, y=-8.870365, z=97.995736, rx=179.999628, ry=2.000598, rz=-0.000236, shoulder=lefty, elbow=epositive, wrist=wpositive, fatherId=frmaster[2]}
  [646] = {x=66.934369, y=-7.885327, z=97.996162, rx=179.999534, ry=1.99962, rz=-0.000284, shoulder=lefty, elbow=epositive, wrist=wpositive, fatherId=frmaster[2]}
  [647] = {x=66.940182, y=-6.897878, z=97.996932, rx=-179.999912, ry=2.000448, rz=0.000178, shoulder=lefty, elbow=epositive, wrist=wpositive, fatherId=frmaster[2]}
  [648] = {x=66.935065, y=-5.914775, z=97.992941, rx=-179.999708, ry=2.000358, rz=0.000311, shoulder=lefty, elbow=epositive, wrist=wpositive, fatherId=frmaster[2]}
  [649] = {x=66.937386, y=-4.927717, z=97.993507, rx=-179.99946, ry=2.000267, rz=0.000366, shoulder=lefty, elbow=epositive, wrist=wpositive, fatherId=frmaster[2]}
  [650] = {x=66.938825, y=-3.941496, z=97.99871, rx=179.999841, ry=2.000494, rz=0.000378, shoulder=lefty, elbow=epositive, wrist=wpositive, fatherId=frmaster[2]}
  [651] = {x=66.938957, y=-2.955069, z=97.999177, rx=-179.999913, ry=2.000391, rz=0.00032, shoulder=lefty, elbow=epositive, wrist=wpositive, fatherId=frmaster[2]}
  [652] = {x=66.938224, y=-1.969743, z=97.994966, rx=-179.99967, ry=2.000275, rz=0.000225, shoulder=lefty, elbow=epositive, wrist=wpositive, fatherId=frmaster[2]}
  [653] = {x=66.936381, y=-0.984542, z=97.995434, rx=-179.999426, ry=2.000161, rz=0.000053, shoulder=lefty, elbow=epositive, wrist=wpositive, fatherId=frmaster[2]}
  [654] = {x=66.933781, y=-0.000734, z=97.991281, rx=-179.999185, ry=2.000036, rz=0.000845, shoulder=lefty, elbow=epositive, wrist=wpositive, fatherId=frmaster[2]}
  [655] = {x=66.939282, y=0.984949, z=98.001068, rx=179.999212, ry=2.000569, rz=-0.000416, shoulder=lefty, elbow=epositive, wrist=wpositive, fatherId=frmaster[2]}
  [656] = {x=66.933979, y=1.969447, z=97.991905, rx=-179.999606, ry=2.000103, rz=0.00027, shoulder=lefty, elbow=epositive, wrist=wpositive, fatherId=frmaster[2]}
  [657] = {x=66.936836, y=2.955565, z=97.996688, rx=179.999733, ry=2.000297, rz=-0.000097, shoulder=lefty, elbow=epositive, wrist=wpositive, fatherId=frmaster[2]}
  [658] = {x=66.937664, y=3.943719, z=97.991806, rx=-179.999042, ry=1.999825, rz=0.000473, shoulder=lefty, elbow=epositive, wrist=wpositive, fatherId=frmaster[2]}
  [659] = {x=66.938423, y=4.928638, z=97.991695, rx=-179.999708, ry=2.000002, rz=0.000033, shoulder=lefty, elbow=epositive, wrist=wpositive, fatherId=frmaster[2]}
  [660] = {x=66.938379, y=5.912498, z=97.996325, rx=179.999629, ry=2.000185, rz=-0.000485, shoulder=lefty, elbow=epositive, wrist=wpositive, fatherId=frmaster[2]}
  [661] = {x=66.936913, y=6.896861, z=98.000598, rx=179.998965, ry=2.000361, rz=-0.00004, shoulder=lefty, elbow=epositive, wrist=wpositive, fatherId=frmaster[2]}
  [662] = {x=66.933575, y=7.882821, z=97.995331, rx=-179.999814, ry=1.999869, rz=0.000343, shoulder=lefty, elbow=epositive, wrist=wpositive, fatherId=frmaster[2]}
  [663] = {x=66.938843, y=8.868541, z=97.994807, rx=179.999561, ry=2.000032, rz=-0.000287, shoulder=lefty, elbow=epositive, wrist=wpositive, fatherId=frmaster[2]}
  [664] = {x=66.932814, y=9.855022, z=97.988947, rx=-179.999223, ry=1.999524, rz=0.000022, shoulder=lefty, elbow=epositive, wrist=wpositive, fatherId=frmaster[2]}
  [665] = {x=66.936219, y=10.839269, z=98.002052, rx=179.999214, ry=2.00003, rz=0.00027, shoulder=lefty, elbow=epositive, wrist=wpositive, fatherId=frmaster[2]}
  [666] = {x=66.937085, y=11.826488, z=97.991525, rx=-179.99953, ry=1.999509, rz=-0.000495, shoulder=lefty, elbow=epositive, wrist=wpositive, fatherId=frmaster[2]}
  [667] = {x=66.936791, y=12.813593, z=97.989871, rx=-179.999216, ry=1.999324, rz=-0.000305, shoulder=lefty, elbow=epositive, wrist=wpositive, fatherId=frmaster[2]}
  [668] = {x=66.936395, y=13.797589, z=97.993041, rx=-179.999843, ry=1.999474, rz=-0.000161, shoulder=lefty, elbow=epositive, wrist=wpositive, fatherId=frmaster[2]}
  [669] = {x=66.935903, y=14.781675, z=97.996004, rx=179.999834, ry=2.000498, rz=0.000305, shoulder=lefty, elbow=epositive, wrist=wpositive, fatherId=frmaster[2]}
  [670] = {x=66.94157, y=15.7685, z=97.998628, rx=179.999249, ry=2.000641, rz=-0.000622, shoulder=lefty, elbow=epositive, wrist=wpositive, fatherId=frmaster[2]}
  [671] = {x=66.936216, y=16.75552, z=97.996031, rx=-179.999497, ry=2.000107, rz=0.000388, shoulder=lefty, elbow=epositive, wrist=wpositive, fatherId=frmaster[2]}
  [672] = {x=66.93965, y=17.741359, z=97.998234, rx=179.999916, ry=2.000243, rz=-0.000613, shoulder=lefty, elbow=epositive, wrist=wpositive, fatherId=frmaster[2]}
  [673] = {x=66.933696, y=18.723088, z=98.00031, rx=179.999285, ry=2.000375, rz=0.000348, shoulder=lefty, elbow=epositive, wrist=wpositive, fatherId=frmaster[2]}
  [674] = {x=66.935036, y=19.707585, z=98.002137, rx=179.998697, ry=2.000505, rz=0.000271, shoulder=lefty, elbow=epositive, wrist=wpositive, fatherId=frmaster[2]}
  [675] = {x=66.933808, y=20.695465, z=97.998746, rx=179.999991, ry=1.999957, rz=0.000132, shoulder=lefty, elbow=epositive, wrist=wpositive, fatherId=frmaster[2]}
  [676] = {x=66.94026, y=21.684815, z=97.995156, rx=-179.999617, ry=1.999737, rz=-0.000012, shoulder=lefty, elbow=epositive, wrist=wpositive, fatherId=frmaster[2]}
  [677] = {x=66.938645, y=22.666696, z=97.996524, rx=179.999793, ry=1.999861, rz=-0.0002, shoulder=lefty, elbow=epositive, wrist=wpositive, fatherId=frmaster[2]}
  [678] = {x=66.935029, y=23.650559, z=98.001671, rx=179.999204, ry=1.999984, rz=0.000574, shoulder=lefty, elbow=epositive, wrist=wpositive, fatherId=frmaster[2]}
  [679] = {x=66.937466, y=24.639905, z=97.992687, rx=-179.999468, ry=1.99941, rz=-0.000675, shoulder=lefty, elbow=epositive, wrist=wpositive, fatherId=frmaster[2]}
  [680] = {x=66.940274, y=25.624974, z=97.997522, rx=179.999986, ry=1.999532, rz=-0.000976, shoulder=lefty, elbow=epositive, wrist=wpositive, fatherId=frmaster[2]}
  [681] = {x=66.93431, y=26.607615, z=97.99736, rx=179.999696, ry=2.000501, rz=0.001113, shoulder=lefty, elbow=epositive, wrist=wpositive, fatherId=frmaster[2]}
  [682] = {x=66.934236, y=27.593195, z=97.996989, rx=-179.999913, ry=2.000271, rz=0.000747, shoulder=lefty, elbow=epositive, wrist=wpositive, fatherId=frmaster[2]}
  [683] = {x=66.940699, y=28.582822, z=97.991497, rx=-179.999485, ry=2.000025, rz=-0.000617, shoulder=lefty, elbow=epositive, wrist=wpositive, fatherId=frmaster[2]}
  [684] = {x=66.904723, y=27.595902, z=97.989956, rx=-179.999121, ry=1.999884, rz=-0.000162, shoulder=lefty, elbow=epositive, wrist=wpositive, fatherId=frmaster[2]}
  [685] = {x=66.876118, y=26.610943, z=97.997173, rx=-179.999649, ry=2.000095, rz=0.000246, shoulder=lefty, elbow=epositive, wrist=wpositive, fatherId=frmaster[2]}
  [686] = {x=66.84575, y=25.626544, z=97.990465, rx=-179.999247, ry=1.99994, rz=-0.000334, shoulder=lefty, elbow=epositive, wrist=wpositive, fatherId=frmaster[2]}
  [687] = {x=66.806342, y=24.637279, z=97.992643, rx=-179.999825, ry=2.000132, rz=0.001041, shoulder=lefty, elbow=epositive, wrist=wpositive, fatherId=frmaster[2]}
  [688] = {x=66.782011, y=23.654853, z=97.994601, rx=-179.999372, ry=1.999994, rz=-0.000656, shoulder=lefty, elbow=epositive, wrist=wpositive, fatherId=frmaster[2]}
  [689] = {x=66.748893, y=22.666602, z=97.996555, rx=-179.999907, ry=2.000185, rz=-0.000356, shoulder=lefty, elbow=epositive, wrist=wpositive, fatherId=frmaster[2]}
  [690] = {x=66.713603, y=21.680277, z=97.993382, rx=-179.999504, ry=2.000028, rz=-0.000086, shoulder=lefty, elbow=epositive, wrist=wpositive, fatherId=frmaster[2]}
  [691] = {x=66.685651, y=20.696339, z=97.998995, rx=-179.999996, ry=2.000218, rz=0.000138, shoulder=lefty, elbow=epositive, wrist=wpositive, fatherId=frmaster[2]}
  [692] = {x=66.648689, y=19.706832, z=97.995597, rx=179.999462, ry=2.000388, rz=0.000366, shoulder=lefty, elbow=epositive, wrist=wpositive, fatherId=frmaster[2]}
  [693] = {x=66.61749, y=18.724032, z=97.995932, rx=179.999908, ry=2.000227, rz=0.000523, shoulder=lefty, elbow=epositive, wrist=wpositive, fatherId=frmaster[2]}
  [694] = {x=66.586349, y=17.737406, z=98.001178, rx=179.999415, ry=2.000409, rz=0.000636, shoulder=lefty, elbow=epositive, wrist=wpositive, fatherId=frmaster[2]}
  [695] = {x=66.552868, y=16.75307, z=97.992193, rx=-179.999201, ry=1.999901, rz=0.000726, shoulder=lefty, elbow=epositive, wrist=wpositive, fatherId=frmaster[2]}
  [696] = {x=66.528221, y=15.767384, z=97.997071, rx=179.999403, ry=2.000405, rz=-0.000203, shoulder=lefty, elbow=epositive, wrist=wpositive, fatherId=frmaster[2]}
  [697] = {x=66.492517, y=14.781778, z=97.996772, rx=179.999846, ry=2.000234, rz=-0.000195, shoulder=lefty, elbow=epositive, wrist=wpositive, fatherId=frmaster[2]}
  [698] = {x=66.455606, y=13.795677, z=97.996284, rx=-179.999711, ry=2.000061, rz=0.000776, shoulder=lefty, elbow=epositive, wrist=wpositive, fatherId=frmaster[2]}
  [699] = {x=66.426978, y=12.809707, z=98.000602, rx=179.999835, ry=2.000225, rz=0.000702, shoulder=lefty, elbow=epositive, wrist=wpositive, fatherId=frmaster[2]}
  [700] = {x=66.396311, y=11.825239, z=97.990536, rx=-179.999686, ry=2.00003, rz=-0.000361, shoulder=lefty, elbow=epositive, wrist=wpositive, fatherId=frmaster[2]}
  [701] = {x=66.365154, y=10.838748, z=97.994414, rx=179.999857, ry=2.000185, rz=0.000491, shoulder=lefty, elbow=epositive, wrist=wpositive, fatherId=frmaster[2]}
  [702] = {x=66.33268, y=9.852136, z=97.998063, rx=179.999399, ry=2.000334, rz=0.000305, shoulder=lefty, elbow=epositive, wrist=wpositive, fatherId=frmaster[2]}
  [703] = {x=66.298858, y=8.865493, z=98.001471, rx=179.998939, ry=2.000476, rz=0.000083, shoulder=lefty, elbow=epositive, wrist=wpositive, fatherId=frmaster[2]}
  [704] = {x=66.271679, y=7.883569, z=97.995365, rx=-179.999591, ry=1.999954, rz=-0.000202, shoulder=lefty, elbow=epositive, wrist=wpositive, fatherId=frmaster[2]}
  [705] = {x=66.234992, y=6.897169, z=97.989044, rx=-179.999113, ry=1.999748, rz=0.000509, shoulder=lefty, elbow=epositive, wrist=wpositive, fatherId=frmaster[2]}
  [706] = {x=66.206151, y=5.912758, z=97.996651, rx=-179.999529, ry=1.999888, rz=0.000135, shoulder=lefty, elbow=epositive, wrist=wpositive, fatherId=frmaster[2]}
  [707] = {x=66.177207, y=4.924753, z=97.999883, rx=179.999106, ry=2.000341, rz=-0.000244, shoulder=lefty, elbow=epositive, wrist=wpositive, fatherId=frmaster[2]}
  [708] = {x=66.145325, y=3.941204, z=97.997665, rx=179.999627, ry=2.00013, rz=-0.000684, shoulder=lefty, elbow=epositive, wrist=wpositive, fatherId=frmaster[2]}
  [709] = {x=66.11287, y=2.955435, z=97.99098, rx=-179.999853, ry=1.999912, rz=-0.000161, shoulder=lefty, elbow=epositive, wrist=wpositive, fatherId=frmaster[2]}
  [710] = {x=66.079573, y=1.968668, z=97.998316, rx=179.999727, ry=2.000032, rz=0.000277, shoulder=lefty, elbow=epositive, wrist=wpositive, fatherId=frmaster[2]}
  [711] = {x=66.044576, y=0.982732, z=97.996022, rx=-179.999752, ry=1.999811, rz=-0.000315, shoulder=lefty, elbow=epositive, wrist=wpositive, fatherId=frmaster[2]}
  [712] = {x=66.017592, y=-0.001609, z=97.998416, rx=179.999866, ry=1.999915, rz=0.000049, shoulder=lefty, elbow=epositive, wrist=wpositive, fatherId=frmaster[2]}
  [713] = {x=65.999681, y=-0.987332, z=97.997129, rx=-179.99952, ry=1.999705, rz=-0.000698, shoulder=lefty, elbow=epositive, wrist=wpositive, fatherId=frmaster[2]}
  [714] = {x=65.981988, y=-1.977289, z=97.99638, rx=-179.999853, ry=1.999816, rz=-0.00049, shoulder=lefty, elbow=epositive, wrist=wpositive, fatherId=frmaster[2]}
  [715] = {x=65.96254, y=-2.965885, z=97.995175, rx=179.99981, ry=1.999915, rz=-0.000318, shoulder=lefty, elbow=epositive, wrist=wpositive, fatherId=frmaster[2]}
  [716] = {x=65.941904, y=-3.954566, z=97.998652, rx=179.999475, ry=2.000016, rz=-0.000223, shoulder=lefty, elbow=epositive, wrist=wpositive, fatherId=frmaster[2]}
  [717] = {x=65.928668, y=-4.939686, z=97.997359, rx=-179.99987, ry=1.999789, rz=-0.000198, shoulder=lefty, elbow=epositive, wrist=wpositive, fatherId=frmaster[2]}
  [718] = {x=65.905723, y=-5.929181, z=97.991408, rx=-179.999263, ry=1.99955, rz=-0.000209, shoulder=lefty, elbow=epositive, wrist=wpositive, fatherId=frmaster[2]}
  [719] = {x=65.89058, y=-6.916011, z=97.990026, rx=-179.99956, ry=1.999627, rz=-0.000265, shoulder=lefty, elbow=epositive, wrist=wpositive, fatherId=frmaster[2]}
  [720] = {x=65.875032, y=-7.904973, z=97.998458, rx=179.9992, ry=2.00003, rz=-0.000405, shoulder=lefty, elbow=epositive, wrist=wpositive, fatherId=frmaster[2]}
  [721] = {x=65.857009, y=-8.89057, z=97.996898, rx=179.999849, ry=1.999777, rz=-0.000607, shoulder=lefty, elbow=epositive, wrist=wpositive, fatherId=frmaster[2]}
  [722] = {x=65.838369, y=-9.877924, z=97.995675, rx=-179.999501, ry=1.999521, rz=0.000114, shoulder=lefty, elbow=epositive, wrist=wpositive, fatherId=frmaster[2]}
  [723] = {x=65.819421, y=-10.867992, z=97.994772, rx=-179.999801, ry=1.999577, rz=-0.000209, shoulder=lefty, elbow=epositive, wrist=wpositive, fatherId=frmaster[2]}
  [724] = {x=65.798866, y=-11.856856, z=97.998436, rx=179.9999, ry=1.999629, rz=0.000392, shoulder=lefty, elbow=epositive, wrist=wpositive, fatherId=frmaster[2]}
  [725] = {x=65.785809, y=-12.842021, z=97.997102, rx=179.999639, ry=1.999665, rz=-0.000044, shoulder=lefty, elbow=epositive, wrist=wpositive, fatherId=frmaster[2]}
  [726] = {x=65.763546, y=-13.83303, z=98.001272, rx=179.999338, ry=1.999705, rz=0.000403, shoulder=lefty, elbow=epositive, wrist=wpositive, fatherId=frmaster[2]}
  [727] = {x=65.74979, y=-14.819583, z=98.000412, rx=179.999375, ry=2.00064, rz=0.000086, shoulder=lefty, elbow=epositive, wrist=wpositive, fatherId=frmaster[2]}
  [728] = {x=65.733916, y=-15.807062, z=97.999684, rx=179.999112, ry=2.000658, rz=0.000417, shoulder=lefty, elbow=epositive, wrist=wpositive, fatherId=frmaster[2]}
  [729] = {x=65.716578, y=-16.793724, z=97.999084, rx=179.999798, ry=2.000357, rz=-0.000362, shoulder=lefty, elbow=epositive, wrist=wpositive, fatherId=frmaster[2]}
  [730] = {x=65.69846, y=-17.781669, z=97.998609, rx=179.999532, ry=2.000358, rz=-0.000184, shoulder=lefty, elbow=epositive, wrist=wpositive, fatherId=frmaster[2]}
  [731] = {x=65.678725, y=-18.768349, z=97.998203, rx=-179.999784, ry=2.000039, rz=-0.000115, shoulder=lefty, elbow=epositive, wrist=wpositive, fatherId=frmaster[2]}
  [732] = {x=65.658835, y=-19.758279, z=97.993483, rx=179.999946, ry=2.00002, rz=0.00091, shoulder=lefty, elbow=epositive, wrist=wpositive, fatherId=frmaster[2]}
  [733] = {x=65.646256, y=-20.743029, z=97.998316, rx=179.999722, ry=2.000001, rz=-0.000182, shoulder=lefty, elbow=epositive, wrist=wpositive, fatherId=frmaster[2]}
  [734] = {x=65.623879, y=-21.732758, z=97.98917, rx=-179.999601, ry=1.999649, rz=0.000658, shoulder=lefty, elbow=epositive, wrist=wpositive, fatherId=frmaster[2]}
  [735] = {x=65.609526, y=-22.719202, z=97.994785, rx=-179.999826, ry=1.999615, rz=0.000373, shoulder=lefty, elbow=epositive, wrist=wpositive, fatherId=frmaster[2]}
  [736] = {x=65.594286, y=-23.706618, z=97.995908, rx=179.999946, ry=1.999566, rz=0.000012, shoulder=lefty, elbow=epositive, wrist=wpositive, fatherId=frmaster[2]}
  [737] = {x=65.579181, y=-24.694344, z=97.992514, rx=-179.999988, ry=2.000423, rz=-0.000188, shoulder=lefty, elbow=epositive, wrist=wpositive, fatherId=frmaster[2]}
  [738] = {x=65.5612, y=-25.680516, z=97.994154, rx=-179.999268, ry=2.000045, rz=-0.000778, shoulder=lefty, elbow=epositive, wrist=wpositive, fatherId=frmaster[2]}
  [739] = {x=65.543216, y=-26.670242, z=97.996436, rx=179.999547, ry=2.000273, rz=-0.000419, shoulder=lefty, elbow=epositive, wrist=wpositive, fatherId=frmaster[2]}
  [740] = {x=65.523167, y=-27.657359, z=97.993987, rx=-179.999738, ry=1.999869, rz=-0.000201, shoulder=lefty, elbow=epositive, wrist=wpositive, fatherId=frmaster[2]}
  [741] = {x=65.501566, y=-28.581893, z=97.993369, rx=-179.999946, ry=1.999627, rz=0.000548, shoulder=lefty, elbow=epositive, wrist=wpositive, fatherId=frmaster[2]}
  [742] = {x=65.86315, y=-27.835371, z=98.188275, rx=179.08517, ry=1.777784, rz=0.014669, shoulder=lefty, elbow=epositive, wrist=wpositive, fatherId=frmaster[2]}
  [743] = {x=66.470551, y=-27.739382, z=98.015321, rx=178.591238, ry=1.419182, rz=0.017163, shoulder=lefty, elbow=epositive, wrist=wpositive, fatherId=frmaster[2]}
  [744] = {x=66.538883, y=-27.186185, z=97.656697, rx=178.252905, ry=0.972815, rz=0.014936, shoulder=lefty, elbow=epositive, wrist=wpositive, fatherId=frmaster[2]}
  [745] = {x=67.112643, y=-26.806639, z=96.90027, rx=178.013068, ry=0.225363, rz=0.003713, shoulder=lefty, elbow=epositive, wrist=wpositive, fatherId=frmaster[2]}
  [746] = {x=67.316563, y=-26.792334, z=96.639435, rx=178.000027, ry=-0.000476, rz=-0.000341, shoulder=lefty, elbow=epositive, wrist=wpositive, fatherId=frmaster[2]}
  [747] = {x=66.327634, y=-26.807555, z=96.641871, rx=177.999519, ry=0.000067, rz=0.000374, shoulder=lefty, elbow=epositive, wrist=wpositive, fatherId=frmaster[2]}
  [748] = {x=65.338391, y=-26.818481, z=96.644023, rx=177.99995, ry=0.000286, rz=0.000099, shoulder=lefty, elbow=epositive, wrist=wpositive, fatherId=frmaster[2]}
  [749] = {x=64.350068, y=-26.832489, z=96.642318, rx=178.000064, ry=-0.000408, rz=-0.000432, shoulder=lefty, elbow=epositive, wrist=wpositive, fatherId=frmaster[2]}
  [750] = {x=63.354686, y=-26.848829, z=96.645732, rx=177.999524, ry=0.000091, rz=0.000321, shoulder=lefty, elbow=epositive, wrist=wpositive, fatherId=frmaster[2]}
  [751] = {x=62.368875, y=-26.859832, z=96.644364, rx=177.999932, ry=0.000307, rz=0.000085, shoulder=lefty, elbow=epositive, wrist=wpositive, fatherId=frmaster[2]}
  [752] = {x=61.374143, y=-26.875112, z=96.643675, rx=178.00002, ry=-0.000427, rz=0.000587, shoulder=lefty, elbow=epositive, wrist=wpositive, fatherId=frmaster[2]}
  [753] = {x=60.390499, y=-26.885941, z=96.63825, rx=178.000415, ry=-0.000212, rz=-0.000625, shoulder=lefty, elbow=epositive, wrist=wpositive, fatherId=frmaster[2]}
  [754] = {x=59.399158, y=-26.90078, z=96.643211, rx=177.999843, ry=0.000278, rz=0.000179, shoulder=lefty, elbow=epositive, wrist=wpositive, fatherId=frmaster[2]}
  [755] = {x=58.408023, y=-26.916597, z=96.648786, rx=177.998964, ry=-0.000149, rz=-0.000283, shoulder=lefty, elbow=epositive, wrist=wpositive, fatherId=frmaster[2]}
  [756] = {x=57.417667, y=-26.927849, z=96.644395, rx=178.000278, ry=-0.000284, rz=-0.000459, shoulder=lefty, elbow=epositive, wrist=wpositive, fatherId=frmaster[2]}
  [757] = {x=56.429024, y=-26.940939, z=96.640667, rx=178.000634, ry=-0.000109, rz=-0.000621, shoulder=lefty, elbow=epositive, wrist=wpositive, fatherId=frmaster[2]}
  [758] = {x=55.441816, y=-26.954812, z=96.647246, rx=178.00003, ry=0.00037, rz=-0.000768, shoulder=lefty, elbow=epositive, wrist=wpositive, fatherId=frmaster[2]}
  [759] = {x=54.445264, y=-26.971783, z=96.6493, rx=177.999117, ry=-0.000103, rz=-0.00019, shoulder=lefty, elbow=epositive, wrist=wpositive, fatherId=frmaster[2]}
  [760] = {x=53.459462, y=-26.983454, z=96.646624, rx=177.999451, ry=0.000067, rz=-0.000317, shoulder=lefty, elbow=epositive, wrist=wpositive, fatherId=frmaster[2]}
  [761] = {x=52.465894, y=-26.999184, z=96.644665, rx=177.999768, ry=0.0002, rz=0.000567, shoulder=lefty, elbow=epositive, wrist=wpositive, fatherId=frmaster[2]}
  [762] = {x=51.481619, y=-27.008812, z=96.642436, rx=178.000087, ry=0.00037, rz=-0.000538, shoulder=lefty, elbow=epositive, wrist=wpositive, fatherId=frmaster[2]}
  [763] = {x=50.489286, y=-27.025359, z=96.646212, rx=177.999149, ry=-0.000115, rz=0.000082, shoulder=lefty, elbow=epositive, wrist=wpositive, fatherId=frmaster[2]}
  [764] = {x=49.497796, y=-27.037486, z=96.640093, rx=178.0004, ry=-0.00028, rz=-0.000003, shoulder=lefty, elbow=epositive, wrist=wpositive, fatherId=frmaster[2]}
  [765] = {x=48.508126, y=-27.05177, z=96.64432, rx=177.999733, ry=0.000145, rz=-0.000073, shoulder=lefty, elbow=epositive, wrist=wpositive, fatherId=frmaster[2]}
  [766] = {x=47.519009, y=-27.064521, z=96.643942, rx=178.000013, ry=0.000274, rz=-0.000133, shoulder=lefty, elbow=epositive, wrist=wpositive, fatherId=frmaster[2]}
  [767] = {x=46.531256, y=-27.078275, z=96.644233, rx=178.000286, ry=0.000403, rz=-0.000182, shoulder=lefty, elbow=epositive, wrist=wpositive, fatherId=frmaster[2]}
  [768] = {x=45.534282, y=-27.095228, z=96.64969, rx=177.999309, ry=-0.000131, rz=0.000485, shoulder=lefty, elbow=epositive, wrist=wpositive, fatherId=frmaster[2]}
  [769] = {x=44.548106, y=-27.107262, z=96.650474, rx=177.999568, ry=-0.000006, rz=0.000455, shoulder=lefty, elbow=epositive, wrist=wpositive, fatherId=frmaster[2]}
  [770] = {x=43.56285, y=-27.119032, z=96.646723, rx=177.999819, ry=0.00012, rz=-0.000564, shoulder=lefty, elbow=epositive, wrist=wpositive, fatherId=frmaster[2]}
  [771] = {x=42.569051, y=-27.132446, z=96.638482, rx=178.001013, ry=-0.000076, rz=0.000424, shoulder=lefty, elbow=epositive, wrist=wpositive, fatherId=frmaster[2]}
  [772] = {x=41.577068, y=-27.148219, z=96.640585, rx=178.000282, ry=0.000296, rz=0.000426, shoulder=lefty, elbow=epositive, wrist=wpositive, fatherId=frmaster[2]}
  [773] = {x=40.58464, y=-27.162991, z=96.64774, rx=177.999275, ry=-0.000252, rz=0.000137, shoulder=lefty, elbow=epositive, wrist=wpositive, fatherId=frmaster[2]}
  [774] = {x=39.602934, y=-27.172997, z=96.640657, rx=178.000457, ry=-0.000409, rz=-0.000843, shoulder=lefty, elbow=epositive, wrist=wpositive, fatherId=frmaster[2]}
  [775] = {x=38.604017, y=-27.188897, z=96.638816, rx=178.000656, ry=-0.000359, rz=0.000185, shoulder=lefty, elbow=epositive, wrist=wpositive, fatherId=frmaster[2]}
  [776] = {x=37.615687, y=-27.203106, z=96.647194, rx=177.999894, ry=0.000001, rz=0.000227, shoulder=lefty, elbow=epositive, wrist=wpositive, fatherId=frmaster[2]}
  [777] = {x=36.628185, y=-27.217132, z=96.641493, rx=178.000085, ry=0.000084, rz=0.000275, shoulder=lefty, elbow=epositive, wrist=wpositive, fatherId=frmaster[2]}
  [778] = {x=35.641469, y=-27.230008, z=96.650419, rx=177.999307, ry=0.000438, rz=0.000335, shoulder=lefty, elbow=epositive, wrist=wpositive, fatherId=frmaster[2]}
  [779] = {x=34.646463, y=-27.24566, z=96.645364, rx=177.999474, ry=0.000483, rz=0.000401, shoulder=lefty, elbow=epositive, wrist=wpositive, fatherId=frmaster[2]}
  [780] = {x=33.661271, y=-27.257205, z=96.645286, rx=177.999643, ry=0.000562, rz=0.000478, shoulder=lefty, elbow=epositive, wrist=wpositive, fatherId=frmaster[2]}
  [781] = {x=32.666443, y=-27.270728, z=96.640784, rx=178.000505, ry=-0.000578, rz=0.000253, shoulder=lefty, elbow=epositive, wrist=wpositive, fatherId=frmaster[2]}
  [782] = {x=31.683644, y=-27.283703, z=96.646527, rx=177.999697, ry=-0.000233, rz=-0.000652, shoulder=lefty, elbow=epositive, wrist=wpositive, fatherId=frmaster[2]}
  [783] = {x=30.691889, y=-27.296915, z=96.642648, rx=177.999837, ry=-0.000192, rz=-0.00055, shoulder=lefty, elbow=epositive, wrist=wpositive, fatherId=frmaster[2]}
  [784] = {x=29.701594, y=-27.311633, z=96.649056, rx=177.999004, ry=0.000111, rz=-0.000439, shoulder=lefty, elbow=epositive, wrist=wpositive, fatherId=frmaster[2]}
  [785] = {x=28.711809, y=-27.32513, z=96.641433, rx=178.000094, ry=-0.000111, rz=-0.00032, shoulder=lefty, elbow=epositive, wrist=wpositive, fatherId=frmaster[2]}
  [786] = {x=27.72314, y=-27.338793, z=96.648443, rx=177.999245, ry=0.000186, rz=-0.000191, shoulder=lefty, elbow=epositive, wrist=wpositive, fatherId=frmaster[2]}
  [787] = {x=26.725864, y=-27.354051, z=96.641517, rx=178.000313, ry=-0.000069, rz=0.000944, shoulder=lefty, elbow=epositive, wrist=wpositive, fatherId=frmaster[2]}
  [788] = {x=25.738824, y=-27.366719, z=96.64914, rx=177.999448, ry=0.000223, rz=0.00009, shoulder=lefty, elbow=epositive, wrist=wpositive, fatherId=frmaster[2]}
  [789] = {x=24.7523, y=-27.37824, z=96.642771, rx=178.000511, ry=0.000006, rz=0.000242, shoulder=lefty, elbow=epositive, wrist=wpositive, fatherId=frmaster[2]}
  [790] = {x=23.757673, y=-27.392669, z=96.641577, rx=178.00059, ry=0.000006, rz=0.000403, shoulder=lefty, elbow=epositive, wrist=wpositive, fatherId=frmaster[2]}
  [791] = {x=22.773515, y=-27.405987, z=96.641076, rx=178.000671, ry=0.000042, rz=-0.000428, shoulder=lefty, elbow=epositive, wrist=wpositive, fatherId=frmaster[2]}
  [792] = {x=21.780514, y=-27.419545, z=96.640527, rx=178.000736, ry=0.000041, rz=-0.000252, shoulder=lefty, elbow=epositive, wrist=wpositive, fatherId=frmaster[2]}
  [793] = {x=20.789157, y=-27.435933, z=96.640793, rx=177.999825, ry=0.000286, rz=-0.000068, shoulder=lefty, elbow=epositive, wrist=wpositive, fatherId=frmaster[2]}
  [794] = {x=19.79748, y=-27.447493, z=96.640857, rx=178.000844, ry=0.000037, rz=0.000124, shoulder=lefty, elbow=epositive, wrist=wpositive, fatherId=frmaster[2]}
  [795] = {x=18.807737, y=-27.463116, z=96.641783, rx=177.999917, ry=0.000277, rz=0.000324, shoulder=lefty, elbow=epositive, wrist=wpositive, fatherId=frmaster[2]}
  [796] = {x=17.818403, y=-27.476642, z=96.647725, rx=177.999953, ry=0.000271, rz=0.000531, shoulder=lefty, elbow=epositive, wrist=wpositive, fatherId=frmaster[2]}
  [797] = {x=16.829555, y=-27.488863, z=96.644105, rx=177.999981, ry=0.000265, rz=0.000745, shoulder=lefty, elbow=epositive, wrist=wpositive, fatherId=frmaster[2]}
  [798] = {x=15.842031, y=-27.502852, z=96.641279, rx=178.000002, ry=0.000258, rz=-0.000034, shoulder=lefty, elbow=epositive, wrist=wpositive, fatherId=frmaster[2]}
  [799] = {x=14.855213, y=-27.515981, z=96.643515, rx=178.000016, ry=0.00025, rz=-0.000805, shoulder=lefty, elbow=epositive, wrist=wpositive, fatherId=frmaster[2]}
  [800] = {x=13.859562, y=-27.529277, z=96.645714, rx=178.000014, ry=0.000206, rz=0.00043, shoulder=lefty, elbow=epositive, wrist=wpositive, fatherId=frmaster[2]}
  [801] = {x=12.874254, y=-27.541772, z=96.639172, rx=178.000986, ry=-0.000036, rz=-0.000328, shoulder=lefty, elbow=epositive, wrist=wpositive, fatherId=frmaster[2]}
  [802] = {x=11.880904, y=-27.557234, z=96.647273, rx=177.999997, ry=0.00015, rz=-0.000079, shoulder=lefty, elbow=epositive, wrist=wpositive, fatherId=frmaster[2]}
  [803] = {x=10.888346, y=-27.572927, z=96.641556, rx=177.999974, ry=0.000104, rz=0.000177, shoulder=lefty, elbow=epositive, wrist=wpositive, fatherId=frmaster[2]}
  [804] = {x=9.905022, y=-27.582637, z=96.645076, rx=177.999952, ry=0.000092, rz=-0.00056, shoulder=lefty, elbow=epositive, wrist=wpositive, fatherId=frmaster[2]}
